// Data types/BACnet Enumerations/E_BACNETUNIT
TYPE E_BACNETUNIT:
(
	BACnetUnit_Area_square_meters	:=	0	,
	BACnetUnit_Area_square_feet	:=	1	,
	BACnetUnit_Electrical_milliamperes	:=	2	,
	BACnetUnit_Electrical_amperes	:=	3	,
	BACnetUnit_Electrical_ohms	:=	4	,
	BACnetUnit_Electrical_volts	:=	5	,
	BACnetUnit_Electrical_kilovolts	:=	6	,
	BACnetUnit_Electrical_megavolts	:=	7	,
	BACnetUnit_Electrical_volt_amperes	:=	8	,
	BACnetUnit_Electrical_kilovolt_amperes	:=	9	,
	BACnetUnit_Electrical_megavolt_amperes	:=	10	,
	BACnetUnit_Electrical_volt_amperes_reactive	:=	11	,
	BACnetUnit_Electrical_kilovolt_amperes_reactive	:=	12	,
	BACnetUnit_Electrical_megavolt_amperes_reactive	:=	13	,
	BACnetUnit_Electrical_degrees_phase	:=	14	,
	BACnetUnit_Electrical_power_factor	:=	15	,
	BACnetUnit_Energy_joules	:=	16	,
	BACnetUnit_Energy_kilojoules	:=	17	,
	BACnetUnit_Energy_watt_hours	:=	18	,
	BACnetUnit_Energy_kilowatt_hours	:=	19	,
	BACnetUnit_Energy_btus	:=	20	,
	BACnetUnit_Energy_therms	:=	21	,
	BACnetUnit_Energy_ton_hours	:=	22	,
	BACnetUnit_Enthalpy_joules_per_kilogram_dry_air	:=	23	,
	BACnetUnit_Enthalpy_btus_per_pound_dry_air	:=	24	,
	BACnetUnit_Frequency_cycles_per_hour	:=	25	,
	BACnetUnit_Frequency_cycles_per_minute	:=	26	,
	BACnetUnit_Frequency_hertz	:=	27	,
	BACnetUnit_Humidity_grams_of_water_per_kilogram_dry_air	:=	28	,
	BACnetUnit_Humidity_percent_relative_humidity	:=	29	,
	BACnetUnit_Length_millimeters	:=	30	,
	BACnetUnit_Length_meters	:=	31	,
	BACnetUnit_Length_inches	:=	32	,
	BACnetUnit_Length_feet	:=	33	,
	BACnetUnit_Light_watts_per_square_foot	:=	34	,
	BACnetUnit_Light_watts_per_square_meter	:=	35	,
	BACnetUnit_Light_lumens	:=	36	,
	BACnetUnit_Light_luxes	:=	37	,
	BACnetUnit_Light_foot_candles	:=	38	,
	BACnetUnit_Mass_kilograms	:=	39	,
	BACnetUnit_Mass_pounds_mass	:=	40	,
	BACnetUnit_Mass_tons	:=	41	,
	BACnetUnit_MassFlow_kilograms_per_second	:=	42	,
	BACnetUnit_MassFlow_kilograms_per_minute	:=	43	,
	BACnetUnit_MassFlow_kilograms_per_hour	:=	44	,
	BACnetUnit_MassFlow_pounds_mass_per_minute	:=	45	,
	BACnetUnit_MassFlow_pounds_mass_per_hour	:=	46	,
	BACnetUnit_Power_watts	:=	47	,
	BACnetUnit_Power_kilowatts	:=	48	,
	BACnetUnit_Power_megawatts	:=	49	,
	BACnetUnit_Power_btus_per_hour	:=	50	,
	BACnetUnit_Power_horsepower	:=	51	,
	BACnetUnit_Power_tons_refrigeration	:=	52	,
	BACnetUnit_Pressure_pascals	:=	53	,
	BACnetUnit_Pressure_kilopascals	:=	54	,
	BACnetUnit_Pressure_bars	:=	55	,
	BACnetUnit_Pressure_pounds_force_per_square_inch	:=	56	,
	BACnetUnit_Pressure_centimeters_of_water	:=	57	,
	BACnetUnit_Pressure_inches_of_water	:=	58	,
	BACnetUnit_Pressure_millimeters_of_mercury	:=	59	,
	BACnetUnit_Pressure_centimeters_of_mercury	:=	60	,
	BACnetUnit_Pressure_inches_of_mercury	:=	61	,
	BACnetUnit_Temperature_degrees_Celsius	:=	62	,
	BACnetUnit_Temperature_degrees_Kelvin	:=	63	,
	BACnetUnit_Temperature_degrees_Fahrenheit	:=	64	,
	BACnetUnit_Temperature_degree_days_Celsius	:=	65	,
	BACnetUnit_Temperature_degree_days_Fahrenheit	:=	66	,
	BACnetUnit_Time_years	:=	67	,
	BACnetUnit_Time_months	:=	68	,
	BACnetUnit_Time_weeks	:=	69	,
	BACnetUnit_Time_days	:=	70	,
	BACnetUnit_Time_hours	:=	71	,
	BACnetUnit_Time_minutes	:=	72	,
	BACnetUnit_Time_seconds	:=	73	,
	BACnetUnit_Velocity_meters_per_second	:=	74	,
	BACnetUnit_Velocity_kilometers_per_hour	:=	75	,
	BACnetUnit_Velocity_feet_per_second	:=	76	,
	BACnetUnit_Velocity_feet_per_minute	:=	77	,
	BACnetUnit_Velocity_miles_per_hour	:=	78	,
	BACnetUnit_Volume_cubic_feet	:=	79	,
	BACnetUnit_Volume_cubic_meters	:=	80	,
	BACnetUnit_Volume_imperial_gallons	:=	81	,
	BACnetUnit_Volume_liters	:=	82	,
	BACnetUnit_Volume_us_gallons	:=	83	,
	BACnetUnit_VolumetricFlow_cubic_feet_per_minute	:=	84	,
	BACnetUnit_VolumetricFlow_cubic_meters_per_second	:=	85	,
	BACnetUnit_VolumetricFlow_imperial_gallons_per_minute	:=	86	,
	BACnetUnit_VolumetricFlow_liters_per_second	:=	87	,
	BACnetUnit_VolumetricFlow_liters_per_minute	:=	88	,
	BACnetUnit_VolumetricFlow_us_gallons_per_minute	:=	89	,
	BACnetUnit_Other_degrees_angular	:=	90	,
	BACnetUnit_Other_degrees_Celsius_per_hour	:=	91	,
	BACnetUnit_Other_degrees_Celsius_per_minute	:=	92	,
	BACnetUnit_Other_degrees_Fahrenheit_per_hour	:=	93	,
	BACnetUnit_Other_degrees_Fahrenheit_per_minute	:=	94	,
	BACnetUnit_Other_no_units	:=	95	,
	BACnetUnit_Other_parts_per_million	:=	96	,
	BACnetUnit_Other_parts_per_billion	:=	97	,
	BACnetUnit_Other_percent	:=	98	,
	BACnetUnit_Other_percent_per_second	:=	99	,
	BACnetUnit_Other_per_minute	:=	100	,
	BACnetUnit_Other_per_second	:=	101	,
	BACnetUnit_Other_psi_per_degree_Fahrenheit	:=	102	,
	BACnetUnit_Other_radians	:=	103	,
	BACnetUnit_Other_revolutions_per_minute	:=	104	,
	BACnetUnit_Currency_currency1	:=	105	,
	BACnetUnit_Currency_currency2	:=	106	,
	BACnetUnit_Currency_currency3	:=	107	,
	BACnetUnit_Currency_currency4	:=	108	,
	BACnetUnit_Currency_currency5	:=	109	,
	BACnetUnit_Currency_currency6	:=	110	,
	BACnetUnit_Currency_currency7	:=	111	,
	BACnetUnit_Currency_currency8	:=	112	,
	BACnetUnit_Currency_currency9	:=	113	,
	BACnetUnit_Currency_currency10	:=	114	,
	BACnetUnit_Area_square_inches	:=	115	,
	BACnetUnit_Area_square_centimeters	:=	116	,
	BACnetUnit_Enthalpy_btus_per_pound	:=	117	,
	BACnetUnit_Length_centimeters	:=	118	,
	BACnetUnit_MassFlow_pounds_mass_per_second	:=	119	,
	BACnetUnit_Temperature_delta_degrees_Fahrenheit	:=	120	,
	BACnetUnit_Temperature_delta_degrees_Kelvin	:=	121	,
	BACnetUnit_Electrical_kilohms	:=	122	,
	BACnetUnit_Electrical_megohms	:=	123	,
	BACnetUnit_Electrical_millivolts	:=	124	,
	BACnetUnit_Energy_kilojoules_per_kilogram	:=	125	,
	BACnetUnit_Energy_megajoules	:=	126	,
	BACnetUnit_Entropy_joules_per_degree_Kelvin	:=	127	,
	BACnetUnit_Entropy_joules_per_kilogram_degree_Kelvin	:=	128	,
	BACnetUnit_Frequency_kilohertz	:=	129	,
	BACnetUnit_Frequency_megahertz	:=	130	,
	BACnetUnit_Frequency_per_hour	:=	131	,
	BACnetUnit_Power_milliwatts	:=	132	,
	BACnetUnit_Pressure_hectopascals	:=	133	,
	BACnetUnit_Pressure_millibars	:=	134	,
	BACnetUnit_VolumetricFlow_cubic_meters_per_hour	:=	135	,
	BACnetUnit_VolumetricFlow_liters_per_hour	:=	136	,
	BACnetUnit_Other_kilowatt_hours_per_square_meter	:=	137	,
	BACnetUnit_Other_kilowatt_hours_per_square_foot	:=	138	,
	BACnetUnit_Other_megajoules_per_square_meter	:=	139	,
	BACnetUnit_Other_megajoules_per_square_foot	:=	140	,
	BACnetUnit_Other_watts_per_square_meter_degree_kelvin	:=	141	,
	BACnetUnit_VolumetricFlow_cubic_feet_per_second	:=	142	,
	BACnetUnit_Other_percent_obscuration_per_foot	:=	143	,
	BACnetUnit_Other_percent_obscuration_per_meter	:=	144	,
	BACnetUnit_Electrical_milliohms	:=	145	,
	BACnetUnit_Energy_megawatt_hours	:=	146	,
	BACnetUnit_Energy_kilo_btus	:=	147	,
	BACnetUnit_Energy_mega_btus	:=	148	,
	BACnetUnit_Enthalpy_kilojoules_per_kilogram_dry_air	:=	149	,
	BACnetUnit_Enthalpy_megajoules_per_kilogram_dry_air	:=	150	,
	BACnetUnit_Entropy_kilojoules_per_degree_Kelvin	:=	151	,
	BACnetUnit_Entropy_megajoules_per_degree_Kelvin	:=	152	,
	BACnetUnit_Force_newton	:=	153	,
	BACnetUnit_MassFlow_grams_per_second	:=	154	,
	BACnetUnit_MassFlow_grams_per_minute	:=	155	,
	BACnetUnit_MassFlow_tons_per_hour	:=	156	,
	BACnetUnit_Power_kilo_btus_per_hour	:=	157	,
	BACnetUnit_Time_hundredths_seconds	:=	158	,
	BACnetUnit_Time_milliseconds	:=	159	,
	BACnetUnit_Torque_newton_meters	:=	160	,
	BACnetUnit_Velocity_millimeters_per_second	:=	161	,
	BACnetUnit_Velocity_millimeters_per_minute	:=	162	,
	BACnetUnit_Velocity_meters_per_minute	:=	163	,
	BACnetUnit_Velocity_meters_per_hour	:=	164	,
	BACnetUnit_VolumetricFlow_cubic_meters_per_minute	:=	165	,
	BACnetUnit_Acceleration_meters_per_second_per_second	:=	166	,
	BACnetUnit_Electrical_amperes_per_meter	:=	167	,
	BACnetUnit_Electrical_amperes_per_square_meter	:=	168	,
	BACnetUnit_Electrical_ampere_square_meters	:=	169	,
	BACnetUnit_Electrical_farads	:=	170	,
	BACnetUnit_Electrical_henrys	:=	171	,
	BACnetUnit_Electrical_ohm_meters	:=	172	,
	BACnetUnit_Electrical_siemens	:=	173	,
	BACnetUnit_Electrical_siemens_per_meter	:=	174	,
	BACnetUnit_Electrical_teslas	:=	175	,
	BACnetUnit_Electrical_volts_per_degree_Kelvin	:=	176	,
	BACnetUnit_Electrical_volts_per_meter	:=	177	,
	BACnetUnit_Electrical_webers	:=	178	,
	BACnetUnit_Light_candelas	:=	179	,
	BACnetUnit_Light_candelas_per_square_meter	:=	180	,
	BACnetUnit_Temperature_degrees_Kelvin_per_hour	:=	181	,
	BACnetUnit_Temperature_degrees_Kelvin_per_minute	:=	182	,
	BACnetUnit_Other_joule_seconds	:=	183	,
	BACnetUnit_Other_radians_per_second	:=	184	,
	BACnetUnit_Other_square_meters_per_Newton	:=	185	,
	BACnetUnit_Other_kilograms_per_cubic_meter	:=	186	,
	BACnetUnit_Other_newton_seconds	:=	187	,
	BACnetUnit_Other_newtons_per_meter	:=	188	,
	BACnetUnit_Other_watts_per_meter_per_degree_Kelvin	:=	189	,
	BACnetUnit_micro_siemens	:=	190	,
	BACnetUnit_cubic_feet_per_hour	:=	191	,
	BACnetUnit_us_gallons_per_hour	:=	192	,
	BACnetUnit_kilometers	:=	193	,
	BACnetUnit_micrometers	:=	194	,
	BACnetUnit_grams	:=	195	,
	BACnetUnit_milligrams	:=	196	,
	BACnetUnit_milliliters	:=	197	,
	BACnetUnit_milliliters_per_second	:=	198	,
	BACnetUnit_decibels	:=	199	,
	BACnetUnit_decibels_millivolt	:=	200	,
	BACnetUnit_decibels_volt	:=	201	,
	BACnetUnit_millisiemens	:=	202	,
	BACnetUnit_watt_hours_reactive	:=	203	,
	BACnetUnit_kilowatt_hours_reactive	:=	204	,
	BACnetUnit_megawatt_hours_reactive	:=	205	,
	BACnetUnit_millimeters_of_water	:=	206	,
	BACnetUnit_per_mille	:=	207	,
	BACnetUnit_grams_per_gram	:=	208	,
	BACnetUnit_kilograms_per_kilogram	:=	209	,
	BACnetUnit_grams_per_kilogram	:=	210	,
	BACnetUnit_milligrams_per_gram	:=	211	,
	BACnetUnit_milligrams_per_kilogram	:=	212	,
	BACnetUnit_grams_per_milliliter	:=	213	,
	BACnetUnit_grams_per_liter	:=	214	,
	BACnetUnit_milligrams_per_liter	:=	215	,
	BACnetUnit_micrograms_per_liter	:=	216	,
	BACnetUnit_grams_per_cubic_meter	:=	217	,
	BACnetUnit_milligrams_per_cubic_meter	:=	218	,
	BACnetUnit_micrograms_per_cubic_meter	:=	219	,
	BACnetUnit_nanograms_per_cubic_meter	:=	220	,
	BACnetUnit_grams_per_cubic_centimeter	:=	221	,
	BACnetUnit_becquerels	:=	222	,
	BACnetUnit_kilobecquerels	:=	223	,
	BACnetUnit_megabecquerels	:=	224	,
	BACnetUnit_gray	:=	225	,
	BACnetUnit_milligray	:=	226	,
	BACnetUnit_microgray	:=	227	,
	BACnetUnit_sieverts	:=	228	,
	BACnetUnit_millisieverts	:=	229	,
	BACnetUnit_microsieverts	:=	230	,
	BACnetUnit_microsieverts_per_hour	:=	231	,
	BACnetUnit_decibels_a	:=	232	,
	BACnetUnit_nephelometric_turbidity_unit	:=	233	,
	BACnetUnit_pH	:=	234	,
	BACnetUnit_grams_per_square_meter	:=	235	,
	BACnetUnit_minutes_per_degree_kelvin	:=	236
);
END_TYPE

// Global Variables/BACnet_Globals
{attribute 'Tc2GvlVarNames'}
VAR_GLOBAL
(* ADS read/write buffer for dynamic sized properties *)
	stBACnet_AdsBuffer		: ST_BACnet_GlobalAdsBuffer; (* 8kByte common ADS buffer used by function blocks that access BACnet over ADS *)
(* global linkable BACnet adapter *)
	fbBACnet_Adapter		: FB_BACnet_Adapter;
(* global visible BACnet adapter reference *)
	pBACnet_Adapter			: POINTER TO FB_BACnet_Adapter;
END_VAR
VAR_GLOBAL CONSTANT
(*********************************************
	Data field maximum
**********************************************)
	BACnet_MaxDayEntry			: UINT := 19;
	BACnet_MaxExSchEntries		: UINT := 9;
	BACnet_MaxTimeValues		: UINT := 9;
	BACnet_MaxObjIdList			: UINT := 1999;
	BACnet_MaxLogBufferEntries	: UINT := 499;
	BACnet_MaxDestinationArray	: UINT := 19;

(*********************************************
	error codes
**********************************************)
	BACnet_ERR_NO_ERROR				: UINT := 0;
	BACnet_ERR_NO_VALID_NET_ID		: UINT := 1;
	BACnet_ERR_WRONG_MAPPING		: UINT := 2;
	BACnet_ERR_OPERATIONAL			: UINT := 3;
	BACnet_ERR_NO_ETH_LINK			: UINT := 4;
	BACnet_ERR_NO_GATEWAY			: UINT := 5;
	BACnet_ERR_WOC_TRIGGER_UNSUP	: UINT := 6;
	BACnet_ERR_WOC_DISABLED			: UINT := 7;
	BACnet_ERR_INVALID_OBJECTID		: UINT := 8;
	BACnet_ERR_INVALID_OBJECTTYPE	: UINT := 10;
	BACnet_ERR_INVALID_CYCLETIME	: UINT := 11;
	BACnet_ERR_INVALID_PARAMETER	: UINT := 12;

(* errors with reset 20.. *)
	BACnet_ERR_PERSISTENT_WRITE		: UINT := 20;
	BACnet_ERR_INVALID_ADS_CONN		: UINT := 21;
	BACnet_ERR_CLIENT_TIMEOUT		: UINT := 22;
	BACnet_ERR_CLIENT_SERVICE		: UINT := 23;
	BACnet_ERR_WOC_TRIGGER_ACTIVE	: UINT := 24;
	BACnet_ERR_REVISION_READ		: UINT := 25;
	BACnet_ERR_PERSISTENT_PLC_WRITE	: UINT := 26;

(* ADS connection errors 30.. *)
	BACnet_ERR_ADS_NO_VALID_NET_ID	: UINT := 30; (* missing a valid Net ID *)
	BACnet_ERR_ADS_Data				: UINT := 31; (* ADS data length is wrong *)
	BACnet_ERR_ADS_Read				: UINT := 32; (* ADS read function was aborted *)
	BACnet_ERR_ADS_Write			: UINT := 33; (* ADS write function was aborted *)
	BACnet_ERR_ADS_ObjType			: UINT := 34; (* object type is wrong *)
	BACnet_ERR_ADS_ObjListEmpty		: UINT := 35; (* object list is empty *)
	BACnet_ERR_ADS_DeviceOP			: UINT := 36; (* device is not operational *)
	BACnet_ERR_ADS_NoDevice			: UINT := 37; (* no device object in object info list *)
	BACnet_ERR_ADS_ObjInstance		: UINT := 38; (* object list info is wrong *)
	BACnet_ERR_ADS_AmsPort			: UINT := 39; (* read AMS port is invalid (<1000) *)
	BACnet_ERR_ADS_ObjectId			: UINT := 40; (* object list info is wrong *)
	BACnet_ERR_ADS_LegacyStack		: UINT := 41; (* revision 6 stack detected (service is available from/above revision 9) *)
	BACnet_ERR_ADS_ObjIdMissmatch	: UINT := 42; (* object ID mapped and object list info are different *)
	BACnet_ERR_ADS_BufferSize		: UINT := 43; (* Property data larger than ADS buffer *)
	BACnet_ERR_ADS_SchedData		: UINT := 44; (* Wrong schedule property data *)
	BACnet_ERR_UnknownEventChoice	: UINT := 45; (* Unknown event choice type *)
	BACnet_ERR_UnknownEntryChoice	: UINT := 46; (* Unknown entry choice type *)
	BACnet_ERR_ADS_TooManyObjects	: UINT := 47; (* List of objects are longer than output list size *)
	BACnet_ERR_ADS_WrongEntrySize	: UINT := 48; (* expected entry size dosn't match read size *)
	BACnet_ERR_ADS_RecipientData	: UINT := 49; (* Invalid recipient data, device type expected *)
	BACnet_ERR_ADS_TooManyEntries	: UINT := 50; (* More entries than expected *)
	BACnet_ERR_ADS_NotEnoughEntries	: UINT := 51; (* Property incomplete, missing entries *)
	BACnet_ERR_ADS_Encoding			: UINT := 52; (* String encoding not supported *)
	BACnet_ERR_ADS_NoServerClient	: UINT := 53; (* Given ADS connection is not an server or client connection (expected bClient or bServer) *)
	BACnet_ERR_ADS_NoNotificationSink: UINT := 54; (* Given ADS connection is not an notification sink connection (expected bNSink) *)

(*********************************************
	other definitions
**********************************************)
	BACnet_ADSTimeOut			: TIME := t#15s;
	BACnet_PlcPersisTimeOut		: TIME := t#2m;
	BACnet_STRING_MAXLENGTH     : INT := 256;
	BACnet_ADSBufferSize		: INT := 8191; (* default 8kByte buffer *)

(* ADS index and groups *)
	BACnet_ADSIGRP_GET_OBJECT_LIST						: UDINT := 16#82400000;
	BACnet_ADSIGRP_CLIENT_COM_PARAMETER					: UDINT := 16#84000000;
	BACnet_ADSIGRP_DEV_R_GETADSPORTBYDEVID				: UDINT := 16#80000047; (* Get AMS Port BY Device ID *)
	BACnet_ADSIGRP_NTFSINK_EVENTNTF_CNT					: UDINT := 16#00000001;
	BACnet_ADSIGRP_NTFSINK_COVNTF_CNT					: UDINT := 16#00000002;
	BACnet_ADSIGRP_NTFSINK_EVENTNTF_READ				: UDINT := 16#00000003;
	BACnet_ADSIGRP_NTFSINK_COVNTF_READ					: UDINT := 16#00000004;
	BACnet_ADSIGRP_NTFSINK_EVENTNTF_DELETE				: UDINT := 16#00000005;
	BACnet_ADSIGRP_NTFSINK_COVNTF_DELETE				: UDINT := 16#00000006;
	BACnet_ADSIGRP_NTFSINK_EVENTNTF_INFO				: UDINT := 16#00000007;
	BACnet_ADSIGRP_NTFSINK_COVNTF_INFO					: UDINT := 16#00000008;
	BACnet_ADSIGRP_WRITE_NTFSINK_EVENTNTF_ACK			: UDINT := 16#00000009;
	BACnet_ADSIGRP_NTFSINK_W_EVENTNTF_ACK_BY_SEQUENCE	: UDINT := 16#0000000A;
	BACnet_ADSIGRP_NTFSINK_W_EVENTNTF_ACK_BY_PARAMETER	: UDINT := 16#0000000B;
	BACnet_ADSIGRP_NTFSINK_R_EVENTNTF_READ_BY_SEQUENCE	: UDINT := 16#0000000C;
	BACnet_ADSIGRP_NTFSINK_R_COVNTF_READ_BY_SEQUENCE	: UDINT := 16#0000000D;
	BACnet_ADSIGRP_NTFSINK_R_EVENTNTF_DELETE_BY_SEQUENCE: UDINT := 16#0000000E;
	BACnet_ADSIGRP_NTFSINK_R_COVNTF_DELETE_BY_SEQUENCE	: UDINT := 16#0000000F;


(* Object specifications *)
	arrBACnet_ObjectTypeNameShort : ARRAY[0..BACnetObjectType_ZCount] OF STRING(5) := [
		'AI' (* BACnetObjectType_AnalogInput :=0 *),
		'AO' (* BACnetObjectType_AnalogOutput :=1 *),
		'AV' (* BACnetObjectType_AnalogValue :=2 *),
		'BI' (* BACnetObjectType_BinaryInput :=3 *),
		'BO' (* BACnetObjectType_BinaryOutput :=4 *),
		'BV' (* BACnetObjectType_BinaryValue :=5 *),
		'CAL' (* BACnetObjectType_Calendar :=6 *),
		'CMD' (* BACnetObjectType_Command :=7 *),
		'DEV' (* BACnetObjectType_Device :=8 *),
		'EE' (* BACnetObjectType_EventEnrollment :=9 *),
		'FILE' (* BACnetObjectType_File :=10 *),
		'GROUP' (* BACnetObjectType_Group :=11 *),
		'LOOP' (* BACnetObjectType_Loop :=12 *),
		'MI' (* BACnetObjectType_MultiStateInput :=13 *),
		'MO' (* BACnetObjectType_MultiStateOutput :=14 *),
		'NC' (* BACnetObjectType_NotificationClass :=15 *),
		'PROG' (* BACnetObjectType_Program :=16 *),
		'SCHED' (* BACnetObjectType_Schedule :=17 *),
		'AVG' (* BACnetObjectType_Averaging :=18 *),
		'MV' (* BACnetObjectType_MultiStateValue :=19 *),
		'TLOG' (* BACnetObjectType_TrendLog :=20 *),
		'LP' (* BACnetObjectType_LifeSafetyPoint :=21 *),
		'LZ' (* BACnetObjectType_LifeSafetyZone :=22 *),
		'ACC' (* BACnetObjectType_Accumulator :=23 *),
		'PC' (* BACnetObjectType_PulseConverter :=24 *),
		''] (* BACnetObjectType_ZCount :=25 *);



END_VAR

// Version/Global_Version
// This function has been automatically generated from the project information.
VAR_GLOBAL CONSTANT
	{attribute 'const_non_replaced'}
	{attribute 'linkalways'}
	stLibVersion_Tc2_BACnetRev12 : ST_LibVersion := (iMajor := 2, iMinor := 4, iBuild := 3, iRevision := 0, sVersion := '2.4.3.0');
END_VAR

// POUs/[obsolete]/F_GetVersionTcBACnet
{attribute 'obsolete' := 'F_GetVersionTcBACnet is obsolete, use stLibVersion_Tc2_BACnetRev12 instead!'}
FUNCTION F_GetVersionTcBACnet : UINT		(* Gets the library version info *)
VAR_INPUT
	nVersionElement		: INT;
END_VAR


(* Possible nVersionElement number:
	1	:	major number
	2	:	minor number
	3	: 	revision number
*)

(* Version history:
Date		|	Version/Author			|	Created with				|	Remark
-----------------------------------------------------------------------------------------------------------------------------------
13/03/12	|	1.0.0	/ MAr			|	V2.11.0 (Build 2218)		|	* Renamed BACnet-datatype ENUM entries
20/03/12	|	1.1.0	/ MAr			|	V2.11.0 (Build 2219)		|	* Added new function blocks with ADS property write support (for WOC on local objects present_value)
			|							|								|	* Added optional input to FB_BACnet_Device to setup the valid ADS port (default 1000)
20/03/12	|	1.1.1	/ MAr			|	V2.11.0 (Build 2219)		|	* Removed obsolete flags in FB_BACnet_Program function block
27/03/12	|	1.1.2	/ MAr			|	V2.11.0 (Build 2219)		|	* FB_BACnet_ReadProp returns real processed data len (nProcessedLen)
			|							|								|	* new helper function "F_BACnet_GetObjId" added
28/03/12	|	1.1.3	/ MAr			|	V2.11.0 (Build 2219)		|	* fixed error reset in "FB_BACnet_Device"
			|							|								|	* filter object instance number in "F_BACnet_GetObjId" to prevent overflow
			|							|								|	* added ending element of BACnetObjectType-Enumeration
			|							|								|	* renamed "bErrorId" to "nErrorId" in "FB_BACnet_NotificationSinkDelEntry"
10/04/12	|	1.1.4	/ MAr			|	V2.11.0 (Build 2220)		|	* FB_BACnet_ReadProp extended with automatic handling for range properties (READ_RANGE)
21/05/12	|	1.2.0	/ MAr			|	V2.11.0 (Build 2222)		|	* Changed ENUM names to capital letter (upper case)
			|							|								|	* Renamed LOOP object process data "_SystemStatus" to "_PresentValueI"
			|							|								|	* Append update logic for remote device into remote object FBs (no need to call remote device FB explicit)
29/05/12	|	1.2.1	/ MAr			|	V2.11.0 (Build 2223)		|	* Append local object for Accumulator access (and also _EX version)
20/07/12	|	1.2.2	/ MAr			|	V2.11.0 (Build 2224)		|	* New kind of BACnet FBs "_RAW" for read/write raw values in PLC program instead of direct hardware link
			|							|								|	* Added "AckedTransitions" flags to "_EX" function blocks
			|							|								|	* Added automatic client reset to FB_BACnet_RemoteDevice (timeouts will counted, but didn't interrupt client functionality if auto-reset is active)
			|							|								|	* New time out counter as output status to FB_BACnet_RemoteDevice added
23/07/12	|	1.2.3	/ MAr			|	V2.11.0 (Build 2226)		|	* Added service fail counter to FB_BACnet_RemoteDevice
20/12/12	|	1.3.0	/ MAr	(Beta)	|	V2.11.0 (Build 2232)		|	* Added ADS-Connection blocks (easy to connect objects over ADS)
			|							|								|	* Added local object function blocks with revision 9 features (BETA versions!)
			|							|								|	* Major-change in exisiting object: FB_BACnet_Loop object dosn't write "OutOfService" anymore
			|							|								|	* New raw version of the ACC object type
			|							|								|	* Added flag helper functions
20/12/12	|	1.3.1	/ MAr	(Beta)	|	V2.11.0 (Build 2232)		|	* Optimized error handling for remote device
			|							|								|	* auto detect legacy mode in remote device and fill AdsConn infos from remote device inputs
08/07/13	|	1.3.2	/ MAr	(Beta)	|	V2.11.0 (Build 2234)		|	* added missing _RAW types to R9
21/08/13	|	1.3.3	/ MAr			|	V2.11.0 (Build 2234)		|	* added new function block for time synchronization over BACnet (local time --> BACnet server --> BACnet broadcast)
06/09/13	|	2.0.0	/ MAr			|	V2.11.0 (Build 2234)		|	* removed legacy function blocks and replaced with R9 versions
			|							|								|	* added function blocks for property access
			|							|								|	* error codes are complete global now
			|							|								|	* optimized process data (removed object ID for basic FBs, sorted process data with focus on alignment)
10/09/13	|	2.0.1	/ MAr			|	V2.11.0 (Build 2237)		|	* new function block for EE object add
02/10/13	|	2.0.2	/ MAr			|	V2.11.0 (Build 2237)		|	* Mapped LocalTime and -Date into Device object
			|							|								|	* Added some helper and signal functions
			|							|								|	* PID auto tuning added into LOOP_EX version
			|							|								|	* Added LOOP objects using internal stack LOOP controller (performance optimized)
			|							|								|	* Removed obsolete function blocks
05/11/13	|	2.0.3	/ MAr			|	V2.11.0 (Build 2237)		|	* Added Multi-State objects as RAW-type
			|							|								|	* Renamed BACnetInfo structure member
			|							|								|	* Added feedback and error flag to RAW function blocks
			|							|								|	* First cycle flag moved on first position in function block logic
			|							|								|	* added WOC-disable service and PLC-startup flag into device object
			|							|								|	* clear data buffer in ReadProp function block (because client data optimized and size of read data maybe lower than buffer size)
19/03/14	|	2.0.4	/ MAr			|	V2.11.0 (Build 2240)		|	* removed obsolete check
10/04/14	|	2.1.0	/ MAr			|	V2.11.0 (Build 2241)		|	* PLC ready flag delayed by device status
23/04/14	|	2.2.0	/ MAr			|	V2.11.0 (Build 2241)		|	* Removed "POLL" version of remote FBs (poll mode can be configured by function block comments)
			|							|								|	* Changed default present_value of object function blocks to "do-nothing"
			|							|								|	  (NULL is furthermore writeable by F_BACnet_RealNull or special Binary-PV [2] or multi-state [0] values)
			|							|								|	* Added new function blocks for PV values (F_BACnet_AnalogPV and F_BACnet_MultiStatePV)
			|							|								|	* Added "a-life" bit to remote device function block
20/05/14	|	2.2.1	/ MAr			|	V2.11.0 (Build 2241)		|	* Fixed "ReadMessageTexts"
			|							|								|	* Default value for command object changed to 0x0 instead 0xffffffff
02/06/14	|	2.2.2	/ MAr			|	V2.11.0 (Build 2241)		|	* Added Notification-Sink read and remove functions (Rev. 12 and above only)
			|							|								|	* Added Notification-Sink function block
			|							|								|	* optimized encoding function (when source and target are diffent memory areas with same byte size)
11/06/14	|	2.2.3	/ MAr			|	V2.11.0 (Build 2241)		|	* Added "bReload" input into local and remote device object
			|							|								|	* automatic LOOP mode detection (ideal mode vs. standard mode) according to the property unit of integral_ and derivative_constant
			|							|								|		- ideal mode means: clear parallel junktion of P, I and D (parameter Kp, Ki and Kd are gain [1] constants for each element)
			|							|								|		- standard mode means: serial junktion of P and I parallel to P and D (parameter Kp is the gain constant [1], Ti and Td are time based [s])
14/11/14	|	2.2.4	/ MAr			|	V2.11.0 (Build 2245)		|	* Added stValidFields into Notification-Event structure
			|							|								|	* Optimized STRING conversion for Object-ID and Date/Time
			|							|								|	* Optimized result type for F_BACnet_GetObjId
20/11/14	|	2.2.5	/ MAr			|	V2.11.0 (Build 2245)		|	* Optimized data handling for Log_Buffer property function block
05/12/14	|	2.2.6	/ MAr			|	V2.11.0 (Build 2245)		|	* Optimized process data default value for remote program object
16/01/15	|	2.2.7	/ MAr			|	V2.11.0 (Build 2245)		|	* New function for "Nothing" process data coding for analog* objects
19/01/15	|	2.3.0	/ MAr			|	V2.11.0	(Build 2245)		|	* Changed default FB to read-only (except local LOOP and PROG)
			|							|								|	* Append new "_WR" function block types to enable write access for commandable basic function blocks (remote and local)
23/01/15	|	2.3.1	/ MAr			|	V2.11.0	(Build 2245)		|	* Optimize value compare in ADS-type of analog* objects
10/02/15	|	2.4.0	/ MAr			|	V2.11.0	(Build 2245)		|	* Remove local _WR-Object types
23/10/15	|	2.4.1	/ MAr			|	V2.11.0 (Build 2248)		|	* Added exception- and weekly-schedule property with REAL value capability
04/11/15	|	2.4.2	/ MAr			|	V2.11.0 (Build 2248)		|	* Fixed data type handling in new REAL type properties
06/11/15	|	2.4.3	/ MAr			|	V2.11.0 (Build 2248)		|	* Fallback for PID mode, if property I or D is deactivated
*)

CASE nVersionElement OF
	1:	F_GetVersionTcBACnet := stLibVersion_Tc2_BACnetRev12.iMajor;
	2:	F_GetVersionTcBACnet := stLibVersion_Tc2_BACnetRev12.iMinor;
	3:	F_GetVersionTcBACnet := stLibVersion_Tc2_BACnetRev12.iBuild;
	4:	F_GetVersionTcBACnet := stLibVersion_Tc2_BACnetRev12.iRevision;
	ELSE
		F_GetVersionTcBACnet := 16#FFFF;
END_CASE

END_FUNCTION

// POUs/BACnet Objects/Local (Server)/FB_BACnet_Device
FUNCTION_BLOCK FB_BACnet_Device
VAR_INPUT
	bReset				: BOOL; (* reset errors *)
	bSupportBackup		: BOOL; (* support backup of PLC persistent data when BACnet backup service is used *)
	bWritePersis		: BOOL; (* Manual trigger for PLC and BACnet persistent data storage *)
	bDisableWOC			: BOOL; (* Deactivate write-on-change mechanism *)
	bReload				: BOOL; (* Reload ADS connection and increase reload counter (trigger autoget) *)
	nAmsPort			: T_AmsPort := 1000; (* default port when port can not be determined automatically *)
END_VAR
VAR_OUTPUT
	nRevision			: DINT := -1; (* protocol revision no. *)
	stAdsConn			: ST_BACnet_AdsConnection;
	eSystemStatus		: E_BACNETDEVICESTATUS;
	bBackupActive		: BOOL;
	bWritePersisActive	: BOOL;
	bOperational		: BOOL;
	bWOCDisabled		: BOOL;
	bFirstCycle			: BOOL;
	dtLocalTime			: ST_BACnet_DateTime;
	bError				: BOOL;
	nErrorId			: UINT;
END_VAR
VAR
	_ObjectId			AT%I*: DWORD;	(* ~(BACnet_ObjectIdentifier:		: LINK) *)
	_LocalDate			AT%I*: DWORD;	(* ~(BACnet_LocalDate		:		: LINK) *)
	_LocalTime			AT%I*: DWORD;	(* ~(BACnet_LocalTime		:		: LINK) *)
	_SystemStatus		AT%I*: WORD;	(* ~(BACnet_SystemStatus	:		: )
								   			(BACnet_ObjectType		: DEV	: )	*)
	_ServerStatus		AT%I*: WORD;	(* ~(BACnet_ServerStatus	:		: )	*)
	_ServerControl		AT%Q*: WORD;	(* ~(BACnet_ServerControl	:		: )	*)
	_fbWritePersistent	: FB_WritePersistentData;
	_rtrigBackup		: R_TRIG;
	_rtrigReset			: R_TRIG;

	_bHasStarted		: BOOL := TRUE;
	_nPlcPort			: T_AmsPort;

	_nUpdateCount	 	: UDINT := 0;
	_nUpdateCountAdp 	: UDINT := 0;
	_BACnetAdapter		: POINTER TO FB_BACnet_Adapter;
	_AdsConn			: _FB_BACnet_AdsConn;
	_WritePersistentProp: FB_BACnet_WriteProp;
	_ReadPersistentProp	: FB_BACnet_ReadProp;
	_iPersis			: INT;
	_nPersistentState	: DWORD;
	_ePersistentState	: E_BACNETPERSISTENTDATASTATE;
	_tonPersisTimeout	: TON;
	_tonPersisPoll		: TON;
	_bPersisWritten		: BOOL;
	_ReadRevisionProp	: FB_BACnet_ReadProp;
	_iRevision			: INT;
	_pLocalDate			: POINTER TO ST_BACnet_Date;
	_pLocalTime			: POINTER TO ST_BACnet_Time;
END_VAR

(* check pointer to bacnet adapter instance *)
IF pBACnet_Adapter > 0 THEN
	_BACnetAdapter := pBACnet_Adapter;
ELSE
	_BACnetAdapter := ADR(fbBACnet_Adapter);
END_IF

(* update adapter *)
IF _BACnetAdapter^._nUpdateCount = _nUpdateCountAdp THEN
	_BACnetAdapter^();
END_IF
(* remind current number of update counter *)
_nUpdateCountAdp := _BACnetAdapter^._nUpdateCount;

(* convert SystemStatus to enumeration *)
eSystemStatus := TO_INT(_SystemStatus);

(* reset trigger *)
_rtrigReset(CLK:= bReset, Q=> );
(* reset error ID and flag *)
IF (nErrorId < 20) OR (nErrorId >= 30) OR _rtrigReset.Q THEN
	nErrorId := BACnet_ERR_NO_ERROR;
END_IF

(* check if NetID is plausible *)
IF _BACnetAdapter^.sAmsNetId = '' THEN
	(* NetId not OK, return with error *)
	nErrorId := BACnet_ERR_NO_VALID_NET_ID;
END_IF

IF ((bSupportBackup) OR (_fbWritePersistent.START AND (_iPersis = 0))) THEN
	(* PLC can be backup't *)
	_ServerControl.0 := TRUE;
ELSE
	(* don't support PLC backup *)
	_ServerControl.0 := FALSE;
	_ServerControl.1 := FALSE;
END_IF

(* trigger backup flag *)
_rtrigBackup(CLK:= (eSystemStatus = BACnetDeviceStatus_BackupInProgress) AND (_iPersis = 0), Q=> );
IF (_iPersis = 0) THEN
	(* only backup if persistent state machine is idle *)
	IF _rtrigBackup.Q AND _ServerControl.0 THEN
		(* trigger backup function *)
		_fbWritePersistent.START := TRUE;
	ELSIF _fbWritePersistent.START AND (NOT _fbWritePersistent.BUSY) THEN
		IF _fbWritePersistent.ERR THEN
			(* backup aborted *)
			nErrorId := BACnet_ERR_PERSISTENT_PLC_WRITE;
		ELSE
			(* backup was successful *)
			_ServerControl.1 := TRUE;
		END_IF
	ELSIF (eSystemStatus <> BACnetDeviceStatus_BackupInProgress) THEN
		(* backup process finished *)
		_ServerControl.1 := FALSE;
	END_IF
END_IF

(* calculate PLC runtime port *)
_nPlcPort := TwinCAT_SystemInfoVarList._AppInfo.AdsPort;

(* call persistent backup *)
_fbWritePersistent(
	NETID	:= '',
	PORT	:= _nPlcPort,
	START	:= ,
	TMOUT	:= BACnet_PlcPersisTimeOut,
	MODE	:= SPDM_VAR_BOOST,
	BUSY	=> ,
	ERR		=> ,
	ERRID	=>
);

(* call ADS connection *)
IF (_ObjectId <> 16#00000000) THEN
	_AdsConn(
		bAutoReload		:= bOperational,
		bReload			:= 	(bReset AND (NOT _AdsConn.bReady))
						OR	bReload,
		bDevOperational	:= bOperational,
		sAmsNetId		:= _BACnetAdapter^.sAmsNetId,
		tDevObjId		:= _ObjectId,
		bIsClient		:= FALSE,
		bReady			=> ,
		bBusy			=> ,
		bDone			=> ,
		bError			=> ,
		nErrorId		=> ,
		stBACnetAds		=> );
END_IF

(* error when ADS connection failed *)
IF _AdsConn.bError THEN
	IF (_AdsConn.nErrorId = BACnet_ERR_ADS_LegacyStack) THEN
		nRevision := 6;
		stAdsConn.bServer := TRUE;
		stAdsConn.bClient := FALSE;
		IF		(NOT stAdsConn.bValid)
			OR	(stAdsConn.nDeviceId <> F_BACnet_GetObjInstance(_ObjectId))
			OR	(stAdsConn.nAmsPort <> nAmsPort)
			OR	(stAdsConn.sAmsNetId <> _BACnetAdapter^.sAmsNetId)
		THEN
			stAdsConn.nReload := stAdsConn.nReload + 1;
		END_IF
		stAdsConn.nDeviceId	:= F_BACnet_GetObjInstance(_ObjectId);
		stAdsConn.sAmsNetId	:= _BACnetAdapter^.sAmsNetId;
		stAdsConn.nAmsPort	:= nAmsPort;
		stAdsConn.bValid	:= TRUE;
	ELSE
		IF (nErrorId = 0) THEN
			nErrorId	:= _AdsConn.nErrorId;
		END_IF
		nRevision := -1;
		stAdsConn	:= _AdsConn.stBACnetAds;
	END_IF
ELSIF _AdsConn.bDone THEN
	stAdsConn := _AdsConn.stBACnetAds;
ELSIF (NOT _AdsConn.bReady) THEN
	nRevision := -1;
END_IF

(* read revision no. *)
_ReadRevisionProp(
	BACnetDevicePort:= stAdsConn.nAmsPort,
	bExecute		:= ,
	sNetId			:= stAdsConn.sAmsNetId,
	ObjectType		:= BACnetObjectType_Device,
	PropertyID		:= BACnetPropertyIdentifier_ProtocolRevision,
	DataType		:= BACnetDataType_UnsignedInteger,
	ObjectInstance	:= stAdsConn.nDeviceId,
	ptrValue		:= ADR(nRevision),
	nLenValue		:= SIZEOF(nRevision),
	bDone			=> ,
	bBusy			=> ,
	bError			=> ,
	nErrID			=> ,
	nProcessedLen	=> );

CASE _iRevision OF

	0: (* idle *)
		IF _AdsConn.bDone THEN
			IF stAdsConn.bValid THEN
				_iRevision := 1;
			END_IF
		END_IF
		_ReadRevisionProp.bExecute := FALSE;

	1: (* read property *)
		IF		_ReadRevisionProp.bExecute
			AND	(NOT _ReadRevisionProp.bBusy)
		THEN
			IF _ReadRevisionProp.bError THEN
				nErrorId := BACnet_ERR_REVISION_READ;
			END_IF
			_ReadRevisionProp.bExecute := FALSE;
			_iRevision := 0;
		ELSE
			_ReadRevisionProp.bExecute := TRUE;
		END_IF

END_CASE


(* Handle persistent data backup *)
_nPersistentState := TO_WORD(_ePersistentState);
_ReadPersistentProp(
	BACnetDevicePort:= stAdsConn.nAmsPort,
	bExecute		:= ,
	sNetId			:= stAdsConn.sAmsNetId,
	ObjectType		:= BACnetObjectType_Device,
	PropertyID		:= 516,
	DataType		:= BACnetDataType_PersistentDataState,
	ObjectInstance	:= F_BACnet_GetObjInstance(_ObjectId),
	ptrValue		:= ADR(_nPersistentState),
	nLenValue		:= SIZEOF(_nPersistentState),
	bDone			=> ,
	bBusy			=> ,
	bError			=> ,
	nErrID			=> ,
	nProcessedLen	=> );

_WritePersistentProp(
	BACnetDevicePort:= stAdsConn.nAmsPort,
	bExecute		:= ,
	sNetId			:= stAdsConn.sAmsNetId,
	ObjectType		:= BACnetObjectType_Device,
	PropertyID		:= 516,
	Priority		:= ,
	DataType		:= BACnetDataType_PersistentDataState,
	ObjectInstance	:= F_BACnet_GetObjInstance(_ObjectId),
	ptrValue		:= ADR(_nPersistentState),
	nLenValue		:= SIZEOF(_nPersistentState),
	bDone			=> ,
	bBusy			=> ,
	bError			=> ,
	nErrID			=> );
_ePersistentState := UDINT_TO_INT(_nPersistentState AND 16#0000FFFF);

CASE _iPersis OF
	0: (* idle *)
		IF		bWritePersis
			AND	(NOT bBackupActive)
			AND	(eSystemStatus <> BACnetDeviceStatus_BackupInProgress)
			AND	(nErrorId = BACnet_ERR_NO_ERROR)
		THEN
			IF stAdsConn.bValid THEN
				_iPersis := 1;
			ELSE
				nErrorId := BACnet_ERR_INVALID_ADS_CONN;
			END_IF
		END_IF
		_ReadPersistentProp.bExecute := FALSE;
		_WritePersistentProp.bExecute := FALSE;
		_bPersisWritten := FALSE;

	1: (* read persistent state machine *)
		IF _ReadPersistentProp.bExecute THEN
			IF _ReadPersistentProp.bError THEN
				_iPersis := 100;
				nErrorId := BACnet_ERR_PERSISTENT_WRITE;
				_ReadPersistentProp.bExecute := FALSE;
			ELSIF (NOT _ReadPersistentProp.bBusy) THEN
				_iPersis := 2;
				_ReadPersistentProp.bExecute := FALSE;
			END_IF
		ELSE
			_ReadPersistentProp.bExecute := TRUE;
		END_IF

	2: (* check state *)
		_tonPersisTimeout.IN := FALSE;
		_tonPersisPoll.IN := FALSE;

		IF _tonPersisPoll.Q THEN
			(* rescan state machine *)
			_iPersis := 1;

		ELSIF _tonPersisTimeout.Q THEN
			(* timeout *)
			_iPersis := 100;
			nErrorId := BACnet_ERR_PERSISTENT_WRITE;

		ELSIF (_ePersistentState = BACnetPersistentData_Disabled) THEN
			_iPersis := 10;

		ELSIF	(_ePersistentState = BACnetPersistentData_Initialize)
			OR	(_ePersistentState >= BACnetPersistentData_Write)
		THEN
			(* wait on idle state *)
			_tonPersisTimeout.IN := TRUE;
			_tonPersisPoll.IN := TRUE;

		ELSIF (_ePersistentState = BACnetPersistentData_NoChange) THEN
			(* start writing PLC *)
			_iPersis := 10;

		ELSIF (_ePersistentState = BACnetPersistentData_Ready) THEN
			IF _bPersisWritten THEN
				(* start writing PLC *)
				_iPersis := 10;
			ELSE
				(* start writing BACnet *)
				_iPersis := 3;
			END_IF

		ELSE
			(* wrong state *)
			_iPersis := 100;
			nErrorId := BACnet_ERR_PERSISTENT_WRITE;
		END_IF
		(* call timer *)
		_tonPersisTimeout(PT:= t#60s, Q=> , ET=> );
		_tonPersisPoll(PT:= t#2s, Q=> , ET=> );

	3: (* write BACnet persistent data *)
		IF _WritePersistentProp.bExecute THEN
			IF _WritePersistentProp.bError THEN
				nErrorId := BACnet_ERR_PERSISTENT_WRITE;
				_iPersis := 100;
				_WritePersistentProp.bExecute := FALSE;
			ELSIF (NOT _WritePersistentProp.bBusy) THEN
				_iPersis := 10; (* start writing PLC *)
				_WritePersistentProp.bExecute := FALSE;
				_bPersisWritten := TRUE;
			END_IF
		ELSE
			_WritePersistentProp.bExecute := TRUE;
			_ePersistentState := BACnetPersistentData_Write;
		END_IF

	10: (* write PLC persistent data *)
		IF _fbWritePersistent.START THEN
			IF _fbWritePersistent.ERR THEN
				(* Aborted *)
				nErrorId := BACnet_ERR_PERSISTENT_PLC_WRITE;
				_iPersis := 100;
				_fbWritePersistent.START := FALSE;
			ELSIF (NOT _fbWritePersistent.BUSY) THEN
				(* Finished *)
				_iPersis := 100;
				_fbWritePersistent.START := FALSE;
			END_IF
		ELSE
			_fbWritePersistent.START := TRUE;
		END_IF

	100:
		IF (NOT bWritePersis) THEN
			_iPersis := 0;
		END_IF

END_CASE

(* control *)
(* Disable write-on-change *)
_ServerControl.2	:= bDisableWOC;
(* PLC running - process data valid *)
_ServerControl.11	:=	(NOT _bHasStarted)
					AND	bOperational;

(* state *)
bWritePersisActive := (_iPersis > 0) AND (_iPersis < 100);
bBackupActive := (eSystemStatus = BACnetDeviceStatus_BackupInProgress);
bOperational :=	(_BACnetAdapter^.eAdapterStatus > BACnetAdapterStatus_Init);
bWOCDisabled := (_ServerStatus AND 16#0004) = 16#0004;
_pLocalDate := ADR(_LocalDate);
_pLocalTime := ADR(_LocalTime);
dtLocalTime.stDate := _pLocalDate^;
dtLocalTime.stTime := _pLocalTime^;

(* update counter *)
IF (_nUpdateCount = 0) AND _bHasStarted THEN
	bFirstCycle := TRUE;
ELSE
	bFirstCycle := FALSE;
END_IF
_bHasStarted := FALSE;
_nUpdateCount := _nUpdateCount + 1;
bError := (nErrorId <> BACnet_ERR_NO_ERROR);

END_FUNCTION_BLOCK

// POUs/BACnet Helper/F_BACnet_GetObjInstance
FUNCTION F_BACnet_GetObjInstance : UDINT
VAR_INPUT
	nObjectId : DWORD;
END_VAR
VAR
END_VAR

F_BACnet_GetObjInstance := nObjectId AND 16#003FFFFF;

END_FUNCTION

// POUs/FB_BACnet_Adapter
FUNCTION_BLOCK FB_BACnet_Adapter
VAR_INPUT
END_VAR
VAR_OUTPUT
	eAdapterStatus		: E_BACNETADAPTERSTATUS;
	bEthLinkOk			: BOOL;
	bGatewayOk			: BOOL;
	sAmsNetId			: T_AmsNetId;
	bFirstCycle			: BOOL;
	bError				: BOOL;
	nErrorId			: UINT;
END_VAR
VAR
	_DeviceStatus	AT%I*: WORD; (* ~(BACnet_DeviceStatus : : ) *)
	_AmsNetId		AT%I*: ARRAY[0..5] OF BYTE; (* ~(BACnet_AmsNetId : : ) *)
	_bHasStarted	: BOOL := TRUE;
	_nUpdateCount	: UDINT := 0;
END_VAR

(* reset error ID *)
nErrorId	:= BACnet_ERR_NO_ERROR;
bError		:= FALSE;

(* update bacnet adapter pointer *)
pBACnet_Adapter := THIS;

(* convert _DeviceStatus to enumeration *)
eAdapterStatus := UINT_TO_INT(SHR((_DeviceStatus AND 16#FF00), 8));

(* update netid *)
UpdateNetID();

(* states *)
bEthLinkOk := (NOT _DeviceStatus.0);
bGatewayOk := (eAdapterStatus = BACnetAdapterStatus_Complete) AND bEthLinkOk;

(* update counter *)
IF (_nUpdateCount = 0) AND _bHasStarted THEN
	bFirstCycle := TRUE;
	_bHasStarted := FALSE;
ELSE
	bFirstCycle := FALSE;
END_IF
_nUpdateCount := _nUpdateCount +1;

ACTION UpdateNetID:
(* read NetId and convert to string *)
sAmsNetId := F_CreateAmsNetId(_AmsNetId);
(* check if it plausible *)
IF sAmsNetId = '0.0.0.0.0.0' THEN
	(* NetId not OK, return with error *)
	bError := TRUE;
	nErrorId := BACnet_ERR_NO_VALID_NET_ID;
	sAmsNetId := '';
END_IF
END_ACTION

END_FUNCTION_BLOCK

// POUs/BACnet ADS/Connection/_FB_BACnet_AdsConn
FUNCTION_BLOCK _FB_BACnet_AdsConn
VAR_INPUT
	bAutoReload			: BOOL := TRUE; (* TRUE --> reload on device operational state and other changes *)
	bReload				: BOOL; (* FALSE --> TRUE refresh information *)
	bIsClient			: BOOL; (* TRUE --> Connection with client device (remote server) *)
END_VAR
VAR_IN_OUT
	bDevOperational		: BOOL;
	sAmsNetId			: T_AmsNetId;
	tDevObjId			: T_BACnet_ObjectIdentifier;
END_VAR
VAR_OUTPUT
	bReady				: BOOL;
	bBusy				: BOOL;
	bDone				: BOOL;
	bError				: BOOL;
	nErrorId			: UINT;
	stBACnetAds			: ST_BACnet_AdsConnection;
END_VAR
VAR
	_BACnetAmsNetID		: T_AmsNetId;
	_fbAdsRead			: FW_AdsRead;
	_arrAdsBuf			: ARRAY[0..13] OF DWORD;
	_rtrigReload		: R_TRIG;
	_rtrigOP			: R_TRIG;
	_i					: INT;
	_nDevObjects		: UDINT;
	_nObjIdx			: UDINT;
	_nAmsPort			: UINT;
	_tObjId				: T_BACnet_ObjectIdentifier := 16#FFFFFFFF;
END_VAR

(*
#define ADSIGRP_BACNET_CLIENT_COM_PARAMETER                      0x010

typedef struct _BACnetDevComData
{
      BACnetObjectIdentifier deviceObjIdentifier;
      BACnetAddress                  netAddress;                      // 10 Byte
      WORD                                 UdpPort;
      DWORD                                IPadress;       
      WORD                                 maxApdu;                         // wird im "Iam" Frame gesetzt
      WORD                                 vendorId;                        // wird im "Iam" Frame gesetzt
      DWORD                                maxSegments;                     // 0 == unspecified number of segments
      DWORD                                segmentTimeout;            // wenn 0 dann Defaultwerte des Devices nehmen 
      DWORD                                apduTimeout;                     // wenn 0 dann Defaultwerte des Devices nehmen
      DWORD                                nApduRetries;              // wenn 0 dann Defaultwerte des Devices nehmen
      BYTE                                 ethernetMacAddr[6];   // Ethernet MAC Address
      BYTE                                 segmentsSupported;         // segmentation both, transmit, receive, no (0 == segmentation both)
      BYTE                                 reserved;
} BACnetDevComData, *PBACnetDevComData;

-----------------------------------------------------
Server:

AdsReadInd, IndexGroup:
#define ADSIGRP_BACNET_GET_OBJECT_LIST                                 0x009

indexOffset == 0 -> Anzahl der Objekte

gerader Index -> Objekttyp
ungerader Index -> ObjetInstanz

IndexOffset 2 sollte daher die DeviceID des Servers sein
*)

(* ads communication *)
_fbAdsRead(
	sNetId		:= _BACnetAmsNetID,
	nPort		:= ,
	nIdxGrp		:= ,
	nIdxOffs	:= ,
	cbReadLen	:= SIZEOF(_arrAdsBuf),
	pReadBuff	:= ADR(_arrAdsBuf),
	bExecute	:= ,
	tTimeout	:= BACnet_ADSTimeOut,
	bBusy		=> ,
	bError		=> ,
	nErrId		=> ,
	cbRead		=> );

(* catch reload event trigger *)
_rtrigReload(CLK:= bReload, Q=> );
_rtrigOP(CLK:= bDevOperational, Q=> );

(* state machine *)
CASE _i OF

	0: (* Idle *)
		IF sAmsNetId = '' THEN
			(* NetId not OK, return with error *)
			nErrorId := BACnet_ERR_ADS_NO_VALID_NET_ID;
			stBACnetAds.bValid := FALSE;
			_BACnetAmsNetID := '';
		ELSIF (F_BACnet_GetObjType(tDevObjId) <> BACnetObjectType_Device) THEN
			(* Object type is not device *)
			nErrorId := BACnet_ERR_ADS_ObjectId;
			stBACnetAds.bValid := FALSE;
			_tObjId := 0;
		ELSIF	_rtrigReload.Q
			OR	(		(		(sAmsNetId <> stBACnetAds.sAmsNetId)
							OR	(tDevObjId <> _tObjId)
							OR	(_BACnetAmsNetID <> sAmsNetId)
							OR	_rtrigOP.Q
						)
					AND	bAutoReload
				)
		THEN
			IF (NOT bDevOperational) THEN
				(* BACnet adapter error *)
				nErrorId := BACnet_ERR_ADS_DeviceOP;
				stBACnetAds.bValid := FALSE;
			ELSE
				nErrorId := BACnet_ERR_NO_ERROR;
				_i := 1;
				(* store connection info *)
				_BACnetAmsNetID	:= sAmsNetId;
				_tObjId := tDevObjId;
			END_IF
		END_IF
		bDone := FALSE;

	(* Determin the AMS port *)
	1:
		IF _fbAdsRead.bExecute THEN
			IF _fbAdsRead.bError THEN
				IF ((UDINT_TO_DWORD(_fbAdsRead.nErrId) AND 16#0000FFFF) = 16#0703) THEN
					(* couldn't read service for AMS port of the device - maybe R6 stack running *)
					nErrorId := BACnet_ERR_ADS_LegacyStack;
				ELSE
					nErrorId := BACnet_ERR_ADS_Read;
				END_IF
				_fbAdsRead.bExecute := FALSE;
				_i := 100;
				stBACnetAds.bValid := FALSE;
			ELSIF (NOT _fbAdsRead.bBusy) THEN
				_fbAdsRead.bExecute := FALSE;
				(* check if port info is valid *)
				IF (_fbAdsRead.cbRead = 2) THEN
					_nAmsPort := DWORD_TO_UINT(_arrAdsBuf[0] AND 16#0000FFFF);
					(* length ok? *)
					IF _nAmsPort >= 1000 THEN
						IF bIsClient THEN
							_i := 100;
							stBACnetAds.nDeviceId := F_BACnet_GetObjInstance(tDevObjId);
						ELSE
							_i := 11;
						END_IF
					ELSE
						(* wrong length, abort *)
						_i := 100;
						nErrorId := BACnet_ERR_ADS_AmsPort;
						stBACnetAds.bValid := FALSE;
					END_IF
				ELSE
					nErrorId := BACnet_ERR_ADS_Data;
					_i := 100;
					stBACnetAds.bValid := FALSE;
				END_IF
			END_IF
		ELSE
			(* start ADS reading *)
			_fbAdsRead.bExecute := TRUE;
			_fbAdsRead.nIdxGrp := BACnet_ADSIGRP_DEV_R_GETADSPORTBYDEVID;
			_fbAdsRead.nPort := 65535;
			_fbAdsRead.nIdxOffs := tDevObjId;
		END_IF

	(* try READ server info -object list length- *)
	11:
		IF _fbAdsRead.bExecute THEN
			IF _fbAdsRead.bError THEN
				_fbAdsRead.bExecute := FALSE;
				_i := 100;
				nErrorId := BACnet_ERR_ADS_Read;
				stBACnetAds.bValid := FALSE;
			ELSIF (NOT _fbAdsRead.bBusy) THEN
				_fbAdsRead.bExecute := FALSE;
				(* check if object list is valid *)
				IF (_fbAdsRead.cbRead = 4) THEN
					_nDevObjects := _arrAdsBuf[0];
					(* length ok? *)
					IF _nDevObjects >= 1 THEN
						_i := 12;
						_nObjIdx := 0;
					ELSE
						(* wrong length, abort *)
						_i := 100;
						nErrorId := BACnet_ERR_ADS_ObjListEmpty;
						stBACnetAds.bValid := FALSE;
					END_IF
				ELSE
					nErrorId := BACnet_ERR_ADS_Data;
					_i := 100;
					stBACnetAds.bValid := FALSE;
				END_IF
			END_IF
		ELSE
			(* start ADS reading *)
			_fbAdsRead.bExecute := TRUE;
			_fbAdsRead.nIdxGrp := BACnet_ADSIGRP_GET_OBJECT_LIST;
			_fbAdsRead.nPort := _nAmsPort;
			_fbAdsRead.nIdxOffs := 0;
		END_IF

	(* try READ server info -object type- *)
	12:
		IF _fbAdsRead.bExecute THEN
			IF _fbAdsRead.bError THEN
				_fbAdsRead.bExecute := FALSE;
				_i := 100;
				nErrorId := BACnet_ERR_ADS_Read;
				stBACnetAds.bValid := FALSE;
			ELSIF (NOT _fbAdsRead.bBusy) THEN
				_fbAdsRead.bExecute := FALSE;
				(* check if type is valid *)
				IF (_fbAdsRead.cbRead = 4) THEN
					IF (_arrAdsBuf[0] = INT_TO_DWORD(BACnetObjectType_Device)) THEN
						(* device object found, go on *)
						_i := 13;
					ELSE
						(* wrong object type, next list entry *)
						_i := 12; (* remain in current step *)
						_nObjIdx := _nObjIdx + 1;
					END_IF
				ELSE
					nErrorId := BACnet_ERR_ADS_Data;
					_i := 100;
					stBACnetAds.bValid := FALSE;
				END_IF
			END_IF
		ELSE
			(* start ADS reading *)
			IF _nObjIdx < _nDevObjects THEN
				_fbAdsRead.bExecute := TRUE;
				_fbAdsRead.nIdxGrp := BACnet_ADSIGRP_GET_OBJECT_LIST;
				_fbAdsRead.nIdxOffs := (_nObjIdx * 2) + 2;
				_fbAdsRead.nPort := _nAmsPort;
			ELSE
				(* no device found, abort *)
				nErrorId := BACnet_ERR_ADS_NoDevice;
				_i := 100;
				stBACnetAds.bValid := FALSE;
			END_IF
		END_IF

	(* try READ server info -object instance- *)
	13:
		IF _fbAdsRead.bExecute THEN
			IF _fbAdsRead.bError THEN
				_fbAdsRead.bExecute := FALSE;
				_i := 100;
				nErrorId := BACnet_ERR_ADS_Read;
				stBACnetAds.bValid := FALSE;
			ELSIF (NOT _fbAdsRead.bBusy) THEN
				_fbAdsRead.bExecute := FALSE;
				(* preset done *)
				_i := 100;
				(* check if ID is valid *)
				IF (_fbAdsRead.cbRead = 4) THEN
					IF (_arrAdsBuf[0] <= 16#3FFFFF) THEN
						IF (F_BACnet_GetObjInstance(tDevObjId) = _arrAdsBuf[0]) THEN
							stBACnetAds.nDeviceId := F_BACnet_GetObjInstance(tDevObjId);
						ELSE
							nErrorId := BACnet_ERR_ADS_ObjIdMissmatch;
							stBACnetAds.bValid := FALSE;
						END_IF
					ELSE
						nErrorId := BACnet_ERR_ADS_ObjInstance;
						stBACnetAds.bValid := FALSE;
					END_IF
				ELSE
					nErrorId := BACnet_ERR_ADS_Data;
					stBACnetAds.bValid := FALSE;
				END_IF
			END_IF
		ELSE
			(* start ADS reading *)
			_fbAdsRead.bExecute := TRUE;
			_fbAdsRead.nIdxGrp := BACnet_ADSIGRP_GET_OBJECT_LIST;
			_fbAdsRead.nIdxOffs := (_nObjIdx * 2) + 1;
			_fbAdsRead.nPort := _nAmsPort;
		END_IF

	100: (* Done *)
		bDone := (nErrorId = BACnet_ERR_NO_ERROR);
		IF (NOT bDone) THEN
			stBACnetAds.bValid := FALSE;
		ELSE
			(* set states *)
			stBACnetAds.bServer := (NOT bIsClient);
			stBACnetAds.bClient := bIsClient;
			stBACnetAds.bValid := TRUE;
			(* count update *)
			stBACnetAds.nReload := stBACnetAds.nReload + 1;
		END_IF
		(* remind device AmsNetID and port *)
		stBACnetAds.sAmsNetId	:= _BACnetAmsNetID;
		stBACnetAds.nAmsPort	:= _nAmsPort;
		(* go idle *)
		_i := 0;

END_CASE

(* set error flag *)
bError	:= (nErrorId <> BACnet_ERR_NO_ERROR);
bBusy	:= _i > 0;
bReady	:= (NOT bError) AND ((NOT bBusy) OR bReady);

END_FUNCTION_BLOCK

// POUs/BACnet Helper/F_BACnet_GetObjType
FUNCTION F_BACnet_GetObjType : E_BACNETOBJECTTYPE
VAR_INPUT
	nObjectId : DWORD;
END_VAR
VAR
END_VAR

F_BACnet_GetObjType := TO_INT(SHR((nObjectId AND 16#FFC00000), 22));

END_FUNCTION

// POUs/BACnet ADS/Properties/Common/FB_BACnet_WriteProp
FUNCTION_BLOCK FB_BACnet_WriteProp
VAR_INPUT
	BACnetDevicePort	: UINT := 16#FFFF;
	bExecute			: BOOL;
	sNetId				: T_AmsNetId;
	ObjectType			: E_BACNETOBJECTTYPE;
	PropertyID			: E_BACNETPROPERTYIDENTIFIER;
	Priority			: E_BACNETPRIORITY;
	DataType			: E_BACNETDATATYPES;
	ObjectInstance		: UDINT;
	ptrValue			: POINTER TO BYTE;
	nLenValue			: UDINT; (* byte size of value (SIZEOF) *)
END_VAR
VAR_OUTPUT
	bDone				: BOOL;
	bBusy				: BOOL;
	bError				: BOOL;
	nErrID				: UDINT;
END_VAR
VAR
	_Write				: ADSWRITE;
	_rtrigStart			: R_TRIG;
	_len_data			: UDINT;
	_nPrio 				: UDINT;
	_ptrDWORD			: POINTER TO DWORD;
	_ptrREAL			: POINTER TO REAL;
	_ptrBYTE			: POINTER TO BYTE;
	_dataPointer		: POINTER TO BYTE;
	_dwordVal			: DWORD;
END_VAR

(* catch the start flag *)
	_rtrigStart(Clk:=bExecute);

(* prepare *)
	IF _rtrigStart.Q AND (NOT bBusy) THEN
		_Write(WRITE := FALSE);
		bDone := FALSE;
		bBusy := TRUE;
		bError := FALSE;
		nErrId := 0;
		_nPrio := SHL(INT_TO_UDINT(Priority), 26);
		_len_data := nLenValue; (* in default, take the user given length *)
		_dataPointer := ptrValue;
		CASE DataType OF
			BACnetDataType_Null 				: _len_data := 0; (* set length to zero *)
			BACnetDataType_Bool 				: _len_data := _len_data; (* 1 *)
			BACnetDataType_CharacterStringExt	: _len_data := _len_data; (* 2 *)

			BACnetDataType_UnsignedInteger,
			BACnetDataType_SignedInteger 		: _len_data := MIN(_len_data, 4); (* 4 *)
				IF (_len_data >= 4) THEN
					(* source data type bigger/equal 4 byte --> OK, take first 4 byte *)
					_ptrDWORD := ptrValue;
				ELSE
					(* upgrade data type from less 4 byte to fully double word *)
					_dwordVal := 0;
					_ptrDWORD := ADR(_dwordVal);
					MEMCPY(destAddr:=_ptrDWORD, srcAddr:=ptrValue, n:=_len_data);
					_dataPointer := _ptrDWORD; (* from here on, point to the internal data source *)
					_len_data := SIZEOF(_dwordVal); (* increase size to internal data type length *)
				END_IF
				(* make some plausibility checks *)
				IF	(		ObjectType = BACnetObjectType_MultiStateInput
						OR	ObjectType = BACnetObjectType_MultiStateOutput
						OR	ObjectType = BACnetObjectType_MultiStateValue
					)
				THEN
					IF _ptrDWORD^ = 0 THEN
						(* set data type and data length to NULL operation *)
						_len_data := 0;
					END_IF
				END_IF

			BACnetDataType_Real 				: _len_data := _len_data; (* 4 *)
				_ptrREAL := ptrValue;
				IF (NOT F_BACnet_IsFinite(_ptrREAL^)) THEN
					(* set data type and data length to NULL operation *)
					_len_data := 0;
				END_IF

			BACnetDataType_Double 				: _len_data := _len_data; (* 8 *)
			BACnetDataType_OctetString 			: _len_data := _len_data; (* 8 *)
			BACnetDataType_Enumerated 			: _len_data := _len_data; (* 8 *)
			BACnetDataType_LimitEnable			: _len_data := _len_data; (* 4 *)
			BACnetDataType_BitString 			: _len_data := _len_data; (* 11 *)

			BACnetDataType_BinaryPV				: _len_data := MIN(_len_data, 1); (* 1 *)
				_ptrByte := ptrValue;
				IF		_len_data <= 0
					OR	_ptrByte^ >= 2
				THEN
					_len_data := 0;
				END_IF
		END_CASE
	ELSIF (NOT bExecute) THEN
		bDone := FALSE;
	END_IF

(* execute *)
	IF bBusy THEN
		_Write(	NETID:= sNetId,
				PORT:= BACnetDevicePort,
				IDXGRP:=16#80000000 + INT_TO_UDINT(PropertyID) + _nPrio,
				IDXOFFS:= F_BACnet_GetObjId(ObjectType, ObjectInstance),
				LEN:= _len_data,
				SRCADDR:= _dataPointer,
				WRITE:= TRUE,
				TMOUT:= BACnet_ADSTimeOut);
		IF NOT _Write.Busy THEN
			IF _Write.Err THEN
				nErrID := _Write.ErrId;
				bError := TRUE;
			END_IF
			_Write(WRITE := FALSE);
			bBusy := FALSE;
			bDone := NOT bError;
		END_IF
	END_IF

END_FUNCTION_BLOCK

// POUs/BACnet Helper/Real/F_BACnet_IsFinite
FUNCTION F_BACnet_IsFinite : BOOL
VAR_INPUT
	fValue		: REAL;
END_VAR
VAR
	fArg		: T_Arg;
END_VAR

fArg.cbLen := SIZEOF(fValue);
fArg.eType := ARGTYPE_REAL;
fArg.pData := ADR(fValue);
F_BACnet_IsFinite := IsFinite(fArg);

END_FUNCTION

// POUs/BACnet Helper/F_BACnet_GetObjId
FUNCTION F_BACnet_GetObjId : T_BACnet_ObjectIdentifier
VAR_INPUT
	ObjectType		: E_BACNETOBJECTTYPE;
	ObjectInstance	: UDINT;
END_VAR
VAR
END_VAR

F_BACnet_GetObjId := F_BACnet_GetObjInstance(ObjectInstance) + SHL(INT_TO_UDINT(ObjectType), 22);

END_FUNCTION

// POUs/BACnet ADS/Properties/Common/FB_BACnet_ReadProp
FUNCTION_BLOCK FB_BACnet_ReadProp
VAR_INPUT
	BACnetDevicePort	: UINT := 16#FFFF;
	bExecute			: BOOL;
	sNetId				: T_AmsNetId;
	ObjectType			: E_BACNETOBJECTTYPE;
	PropertyID			: E_BACNETPROPERTYIDENTIFIER;
	DataType			: E_BACNETDATATYPES;
	ObjectInstance		: UDINT;
	ptrValue			: POINTER TO BYTE;
	nLenValue			: UDINT; (* byte size of value (SIZEOF) *)
END_VAR
VAR_OUTPUT
	bDone				: BOOL;
	bBusy				: BOOL;
	bError				: BOOL;
	nErrID				: UDINT;
	nProcessedLen		: UDINT; (* the received data length (can be different to given length) *)
END_VAR
VAR
	_Read				: FW_AdsRead;
	_rtrigStart			: R_TRIG;
	_len_data			: UDINT;
END_VAR

(* catch the start flag *)
	_rtrigStart(Clk:=bExecute);

(* prepare *)
	IF _rtrigStart.Q AND (NOT bBusy) THEN
		_Read(bExecute := FALSE);
		bDone := FALSE;
		bBusy := TRUE;
		bError := FALSE;
		nErrId := 0;
		nProcessedLen := 0;
		(* in default, take the user given length *)
		_len_data := nLenValue;
		(* set index group for read property access *)
		_Read.nIdxGrp := 16#80000000 + INT_TO_UDINT(PropertyID);
		(* handle special data type things *)
		CASE DataType OF
			BACnetDataType_Null 				: _len_data := 0; (* set length to zero *)
			BACnetDataType_Bool 				: _len_data := _len_data; (* 1 *)
			BACnetDataType_CharacterStringExt	: _len_data := _len_data; (* 2 *)
			BACnetDataType_UnsignedInteger 		: _len_data := _len_data; (* 4 *)
			BACnetDataType_SignedInteger 		: _len_data := _len_data; (* 4 *)
			BACnetDataType_Real 				: _len_data := _len_data; (* 4 *)
			BACnetDataType_Double 				: _len_data := _len_data; (* 8 *)
			BACnetDataType_OctetString 			: _len_data := _len_data; (* 8 *)
			BACnetDataType_Enumerated 			: _len_data := _len_data; (* 8 *)
			BACnetDataType_LimitEnable			: _len_data := _len_data; (* 4 *)
			BACnetDataType_BitString 			: _len_data := _len_data; (* 11 *)
			BACnetDataType_LogRecordList:
				_len_data := _len_data; (* n *)
				_Read.nIdxGrp := _Read.nIdxGrp + 16#03800000; (* read range *)
		END_CASE;
	ELSIF (NOT bExecute) THEN
		bDone := FALSE;
	END_IF


(* execute *)
	IF bBusy THEN
		_Read(
			sNetId		:= sNetId,
			nPort		:= BACnetDevicePort,
			nIdxGrp		:= , (* see above *)
			nIdxOffs	:= F_BACnet_GetObjId(ObjectType, ObjectInstance),
			cbReadLen	:= _len_data,
			pReadBuff	:= ptrValue,
			bExecute	:= TRUE,
			tTimeout	:= BACnet_ADSTimeOut,
			bBusy		=> ,
			bError		=> ,
			nErrId		=> ,
			cbRead		=> );
		IF (NOT _Read.bBusy) THEN
			IF _Read.bError THEN
				nErrID := _Read.nErrId;
				bError := TRUE;
				nProcessedLen := 0;
			ELSE
				(* success *)
				nProcessedLen := _Read.cbRead;
				IF (_Read.cbRead < nLenValue) THEN
					(* fill unused part of buffer with zero *)
					MEMSET(destAddr:=(ptrValue+_Read.cbRead), fillByte:=0, n:=(nLenValue-_Read.cbRead));
				END_IF
			END_IF
			_Read(bExecute := FALSE);
			bBusy := FALSE;
			bDone := NOT bError;
		END_IF;
	END_IF

END_FUNCTION_BLOCK

// POUs/BACnet Objects/Local (Server)/FB_BACnet_Program
FUNCTION_BLOCK FB_BACnet_Program
VAR_INPUT
	bRelease			: BOOL;
	bCommonError		: BOOL;
	bWaitForSomething	: BOOL;
	stDoneFlags			: ST_BACnet_ProgramHandshakeRequests;
	stFailedFlags		: ST_BACnet_ProgramHandshakeRequests;
	bModeUnloadComplex	: BOOL := TRUE;
END_VAR
VAR_IN_OUT
	Device				: FB_BACnet_Device;
END_VAR
VAR_OUTPUT
	bReady				: BOOL;
	bOverridden			: BOOL;
	bOutOfService		: BOOL;
	bFault				: BOOL;
	bInAlarm			: BOOL;
	stRequestFlags		: ST_BACnet_ProgramHandshakeRequests;
	stActiveStateFlags	: ST_BACnet_ProgramHandshakeStates;
	bError				: BOOL;
	nErrorId			: UINT;
END_VAR
VAR
(* from BACnet to PLC *)
	_ProgramChange AT%I*: WORD;			(* ~(BACnet_ProgramChange 				:		: )
											(BACnet_ObjectType 					: PROG	: ) *)
	_StatusFlags AT%I*: WORD;			(* ~(BACnet_StatusFlags 				:		: )	*)

(* from PLC to BACnet *)
	_ProgramState AT%Q*: WORD;			(* ~(BACnet_ProgramState 				:		: ) *)
	_ReasonForHalt AT%Q*: WORD;			(* ~(BACnet_ReasonForHalt 				:		: )	*)
	_SetProgramReadyState AT%Q*: BOOL;	(* ~(BACnet_SetProgramReadyState 		:		: )	*)

(* internal signals *)
	_StatusFlagsBits 	: ST_BACnet_StatusFlags;
	_bTriggerSetup		: BOOL;
	_ActiveChange		: E_BACNETPROGRAMREQUEST; (* ACTIVE PROGRAM CHANGE *)
	_bLockedForChange	: BOOL;
	_nUpdateCount		: UDINT := 0;
END_VAR

(* update server device *)
IF (Device._nUpdateCount = _nUpdateCount) THEN
	Device();
END_IF
(* remind current number of update counter *)
_nUpdateCount := Device._nUpdateCount;

(* check BitString format of StatusFlags --> if StatusFlags are less than 4, object isn't linked correctly *)
IF (_StatusFlags < 4) THEN
	(* wrong mapping *)
	nErrorId := BACnet_ERR_WRONG_MAPPING;
	bReady := FALSE;

ELSIF Device.bOperational THEN
	(* ready state *)
	bReady := TRUE;
	nErrorId := BACnet_ERR_NO_ERROR;

	(* decode status flags *)
	_StatusFlagsBits := F_BACnet_StatusFlags(_StatusFlags);

	(* copy states to output *)
	bOverridden := _StatusFlagsBits.overridden;
	bOutOfService := _StatusFlagsBits.out_of_service;
	bFault := _StatusFlagsBits.fault;
	bInAlarm := _StatusFlagsBits.in_alarm;

	(* execute change *)
	CASE _ActiveChange OF
		BACnetProgramRequest_ready:
			(* idle *);

		BACnetProgramRequest_load:
			_ProgramState	 := TO_WORD(BACnetProgramState_loading);
			_ActiveChange	:= BACnetProgramRequest_ready;

		BACnetProgramRequest_restart,
		BACnetProgramRequest_run:
			IF _bTriggerSetup THEN
				(* wait on setup finish *)
				IF stFailedFlags.bSetup OR bCommonError OR (NOT bRelease) THEN
					(* abort *)
					_ProgramState := TO_WORD(BACnetProgramState_halted);
					_ActiveChange := BACnetProgramRequest_ready;
					_ReasonForHalt  := TO_WORD(BACnetProgramError_progerror_internal);
				ELSIF stDoneFlags.bSetup THEN
					(* setup done, start "normal" running mode *)
					_bTriggerSetup := FALSE;
					_ActiveChange := BACnetProgramRequest_run;
				END_IF
			ELSE
				IF stFailedFlags.bRun OR bCommonError OR (NOT bRelease) THEN
					(* abort *)
					_ProgramState := TO_WORD(BACnetProgramState_halted);
					_ActiveChange := BACnetProgramRequest_ready;
					_ReasonForHalt  := TO_WORD(BACnetProgramError_progerror_internal);
				ELSIF stDoneFlags.bRun THEN
					(* switch to running state *)
					_ProgramState  := TO_WORD(BACnetProgramState_running);
					_ActiveChange := BACnetProgramRequest_ready;
				END_IF
			END_IF

		BACnetProgramRequest_halt:
			(* wait on halted *)
			IF stFailedFlags.bHalt OR bCommonError OR (NOT bRelease) THEN
				(* abort *)
				_ProgramState := TO_WORD(BACnetProgramState_halted);
				_ActiveChange := BACnetProgramRequest_ready;
				_ReasonForHalt  := TO_WORD(BACnetProgramError_progerror_internal);
			ELSIF stDoneFlags.bHalt THEN
				(* halted *)
				_ProgramState := TO_WORD(BACnetProgramState_halted);
				_ActiveChange := BACnetProgramRequest_ready;
				_ReasonForHalt  := TO_WORD(BACnetProgramError_program);
			END_IF

		BACnetProgramRequest_unload:
			_ProgramState	 := TO_WORD(BACnetProgramState_unloading);
			_ActiveChange	:= BACnetProgramRequest_ready;

	END_CASE

	(* start change request and handle error states *)
	IF (_ActiveChange = BACnetProgramRequest_ready) THEN

		CASE TO_DINT(_ProgramState) OF
			BACnetProgramState_idle:
				IF bCommonError THEN
					(* abort *)
					_ProgramState := TO_WORD(BACnetProgramState_halted);
					_ReasonForHalt  := TO_WORD(BACnetProgramError_progerror_internal);
				ELSIF (NOT bRelease) THEN
					(* abort *)
					_ProgramState := TO_WORD(BACnetProgramState_halted);
					_ReasonForHalt  := TO_WORD(BACnetProgramError_other);
				ELSIF (NOT _bLockedForChange) THEN
					_ReasonForHalt  := TO_WORD(BACnetProgramError_program_normal);
					CASE TO_DINT(_ProgramChange) OF
						BACnetProgramRequest_unload,
						BACnetProgramRequest_halt:
							(* acknowledge without execution *)
							_SetProgramReadyState	:= TRUE;
						BACnetProgramRequest_restart,
						BACnetProgramRequest_run,
						BACnetProgramRequest_load:
							(* execute request *)
							_ActiveChange := BACnetProgramRequest_load;
							_bTriggerSetup := TRUE;
					END_CASE
				END_IF

			BACnetProgramState_loading:
				IF bCommonError THEN
					(* abort *)
					_ProgramState := TO_WORD(BACnetProgramState_halted);
					_ReasonForHalt  := TO_WORD(BACnetProgramError_progerror_internal);
				ELSIF (NOT bRelease) THEN
					(* abort *)
					_ProgramState := TO_WORD(BACnetProgramState_halted);
					_ReasonForHalt  := TO_WORD(BACnetProgramError_other);
				ELSIF stFailedFlags.bLoad THEN
					(* abort *)
					_ProgramState := TO_WORD(BACnetProgramState_halted);
					_ReasonForHalt  := TO_WORD(BACnetProgramError_load_failed);
				ELSIF stDoneFlags.bLoad THEN
					(* DONE *)
					_bTriggerSetup := TRUE;
					_ActiveChange := BACnetProgramRequest_run;
				ELSIF (NOT _bLockedForChange) THEN
					_ReasonForHalt  := TO_WORD(BACnetProgramError_program_normal);
					CASE to_dint(_ProgramChange) OF
						BACnetProgramRequest_load,
						BACnetProgramRequest_run,
						BACnetProgramRequest_halt,
						BACnetProgramRequest_restart:
							(* acknowledge without execution *)
							_SetProgramReadyState	:= TRUE;
						BACnetProgramRequest_unload:
							(* execute request *)
							_ActiveChange := to_int(_ProgramChange);
					END_CASE
				END_IF

			BACnetProgramState_running:
				IF bCommonError THEN
					(* abort *)
					_ProgramState := TO_WORD(BACnetProgramState_halted);
					_ReasonForHalt  := TO_WORD(BACnetProgramError_progerror_internal);
				ELSIF (NOT bRelease) THEN
					(* abort *)
					_ProgramState := TO_WORD(BACnetProgramState_halted);
					_ReasonForHalt  := TO_WORD(BACnetProgramError_other);
				ELSIF bWaitForSomething THEN
					(* wait on something *)
					_ProgramState  := TO_WORD(BACnetProgramState_waiting);
				ELSIF (NOT _bLockedForChange) THEN
					_ReasonForHalt  := TO_WORD(BACnetProgramError_program_normal);
					CASE to_dint(_ProgramChange) OF
						BACnetProgramRequest_run:
							(* is already running *)
							_SetProgramReadyState	:= TRUE;
						BACnetProgramRequest_unload,
						BACnetProgramRequest_halt:
							(* execute request *)
							_ActiveChange := to_int(_ProgramChange);
						BACnetProgramRequest_restart,
						BACnetProgramRequest_load:
							(* retrigger setup *)
							_ActiveChange := BACnetProgramRequest_restart;
							_bTriggerSetup := TRUE;
					END_CASE
				END_IF

			BACnetProgramState_waiting:
				IF bCommonError THEN
					(* abort *)
					_ProgramState := TO_WORD(BACnetProgramState_halted);
					_ReasonForHalt  := TO_WORD(BACnetProgramError_progerror_internal);
				ELSIF (NOT bRelease) THEN
					(* abort *)
					_ProgramState := TO_WORD(BACnetProgramState_halted);
					_ReasonForHalt  := TO_WORD(BACnetProgramError_other);
				ELSIF (NOT bWaitForSomething) THEN
					(* got it *)
					_ProgramState  := TO_WORD(BACnetProgramState_running);
				ELSIF (NOT _bLockedForChange) THEN
					_ReasonForHalt  := TO_WORD(BACnetProgramError_program_normal);
					CASE to_dint(_ProgramChange) OF
						BACnetProgramRequest_run:
							(* is already running *)
							_SetProgramReadyState	:= TRUE;
						BACnetProgramRequest_unload,
						BACnetProgramRequest_halt:
							(* execute request *)
							_ActiveChange := to_int(_ProgramChange);
					END_CASE
				END_IF

			BACnetProgramState_halted:
				IF (NOT bCommonError) AND bRelease AND (NOT _bLockedForChange) THEN
					CASE TO_DINT(_ProgramChange) OF
						BACnetProgramRequest_halt:
							(* acknowledge without execution *)
							_SetProgramReadyState	:= TRUE;
						BACnetProgramRequest_unload:
							(* execute request *)
							_ActiveChange := TO_INT(_ProgramChange);
						BACnetProgramRequest_restart,
						BACnetProgramRequest_load:
							(* retrigger setup *)
							_ActiveChange := BACnetProgramRequest_restart;
							_bTriggerSetup := TRUE;
						BACnetProgramRequest_run:
							(* start, but don't trigger setup *)
							_ActiveChange := TO_INT(_ProgramChange);
							_bTriggerSetup := FALSE;
					END_CASE
				END_IF

			BACnetProgramState_unloading:
				IF bModeUnloadComplex THEN
					_ReasonForHalt  := TO_WORD(BACnetProgramError_program_normal);
					IF bCommonError THEN
						(* abort *)
						_ProgramState := TO_WORD(BACnetProgramState_halted);
						_ActiveChange := BACnetProgramRequest_ready;
						_ReasonForHalt  := TO_WORD(BACnetProgramError_progerror_internal);
					ELSIF (NOT bRelease) THEN
						(* abort *)
						_ProgramState := TO_WORD(BACnetProgramState_halted);
						_ActiveChange := BACnetProgramRequest_ready;
						_ReasonForHalt  := TO_WORD(BACnetProgramError_other);
					ELSIF stFailedFlags.bUnload THEN
						(* abort *)
						_ProgramState := TO_WORD(BACnetProgramState_halted);
						_ActiveChange := BACnetProgramRequest_ready;
						_ReasonForHalt  := TO_WORD(BACnetProgramError_other);
					ELSIF stDoneFlags.bUnload THEN
						(* DONE *)
						_ActiveChange := BACnetProgramRequest_ready;
						_ProgramState  := TO_WORD(BACnetProgramState_idle);
					ELSIF (NOT _bLockedForChange) THEN
						CASE TO_DINT(_ProgramChange) OF
							BACnetProgramRequest_load,
							BACnetProgramRequest_run,
							BACnetProgramRequest_halt,
							BACnetProgramRequest_restart,
							BACnetProgramRequest_unload:
								(* acknowledge without execution *)
								_SetProgramReadyState	:= TRUE;
						END_CASE
					END_IF
				END_IF

		END_CASE
	END_IF

	(* check state of "change" request *)
	IF (_ActiveChange <> BACnetProgramRequest_ready) THEN
		(* request is active, lock execution *)
		_bLockedForChange		:= TRUE;
	ELSIF _bLockedForChange AND (NOT _SetProgramReadyState) THEN
		(* change finished, tell the stack done *)
		_SetProgramReadyState	:= TRUE;
		_bTriggerSetup			:= FALSE;
	ELSIF (TO_INT(_ProgramChange) = BACnetProgramRequest_ready) THEN
		(* wait on new requests *)
		_SetProgramReadyState	:= FALSE;
		_bLockedForChange		:= FALSE;
		_bTriggerSetup			:= FALSE;
	ELSE
		(* new request *)
		_bTriggerSetup			:= FALSE;
	END_IF

	(* external requests *)
	stRequestFlags.bLoad			:= _ProgramState = TO_WORD(BACnetProgramState_loading) AND (NOT _bLockedForChange);
	stRequestFlags.bSetup			:=	(		(_ActiveChange = BACnetProgramRequest_run)
										OR	(_ActiveChange = BACnetProgramRequest_restart)
									)
								AND	_bTriggerSetup;
	stRequestFlags.bRun			:= (_ActiveChange = BACnetProgramRequest_run) AND (NOT _bTriggerSetup);
	stRequestFlags.bHalt			:= _ActiveChange = BACnetProgramRequest_halt;
	stRequestFlags.bUnload		:=	(_ActiveChange = BACnetProgramRequest_unload)
								OR	(		_ProgramState = TO_WORD(BACnetProgramState_unloading)
										AND	(NOT _bLockedForChange)
									);

	(* active status flags *)
	stActiveStateFlags.bIdle		:= _ProgramState = TO_WORD(BACnetProgramState_idle);
	stActiveStateFlags.bLoading		:= _ProgramState = TO_WORD(BACnetProgramState_loading);
	stActiveStateFlags.bRunning		:= _ProgramState = TO_WORD(BACnetProgramState_running);
	stActiveStateFlags.bWaiting		:= _ProgramState = TO_WORD(BACnetProgramState_waiting);
	stActiveStateFlags.bHalted		:= _ProgramState = TO_WORD(BACnetProgramState_halted);
	stActiveStateFlags.bUnloading	:= _ProgramState = TO_WORD(BACnetProgramState_unloading);
ELSE
	(* server device not ready, reset local ready also *)
	bReady := FALSE;
	nErrorId := BACnet_ERR_OPERATIONAL;
END_IF
(* set error flag *)
bError := (nErrorId <> BACnet_ERR_NO_ERROR);

END_FUNCTION_BLOCK

// POUs/BACnet Helper/Flags/F_BACnet_StatusFlags
FUNCTION F_BACnet_StatusFlags : ST_BACnet_StatusFlags
VAR_INPUT
	data	: WORD;
END_VAR
VAR
END_VAR

F_BACnet_StatusFlags.in_alarm:= _F_BACnet_IsBitFieldBitSet( data:=data, bitNbr:=BACnetStatusFlags_in_alarm);
F_BACnet_StatusFlags.fault:= _F_BACnet_IsBitFieldBitSet( data:=data, bitNbr:=BACnetStatusFlags_fault);
F_BACnet_StatusFlags.overridden:= _F_BACnet_IsBitFieldBitSet( data:=data, bitNbr:=BACnetStatusFlags_overridden);
F_BACnet_StatusFlags.out_of_service:= _F_BACnet_IsBitFieldBitSet( data:=data, bitNbr:=BACnetStatusFlags_out_of_service);

END_FUNCTION

// POUs/BACnet Helper/[internal]/_F_BACnet_IsBitFieldBitSet
FUNCTION _F_BACnet_IsBitFieldBitSet : BOOL
VAR_INPUT
	data	:	DWORD;
	bitNbr		:	INT;
END_VAR
VAR
END_VAR

_F_BACnet_IsBitFieldBitSet:= (data AND (SHR(DWORD#16#00008000,_F_BACnet_BitFieldBit(bitNbr)))) > 0;

END_FUNCTION

// POUs/BACnet Helper/[internal]/_F_BACnet_BitFieldBit
FUNCTION _F_BACnet_BitFieldBit : WORD
VAR_INPUT
	bitNbr	:	INT;
END_VAR
VAR
END_VAR

_F_BACnet_BitFieldBit := to_word((bitNbr/8) * 8 + (bitNbr MOD 8));

END_FUNCTION

// POUs/BACnet ADS/[obsolete]/FB_BACnet_NotificationSinkDelEntry
FUNCTION_BLOCK FB_BACnet_NotificationSinkDelEntry
VAR_INPUT
	bExecute	: BOOL;
	nIndex		: UDINT;
	sNetId		: T_AmsNetId;
	nPort		: T_AmsPort;
	tTimeout	: TIME := BACnet_ADSTimeOut;
END_VAR
VAR_OUTPUT
	bBusy		: BOOL;
	bEmpty		: BOOL;
	bError		: BOOL;
	nErrorId	: UDINT;
END_VAR
VAR
	_AdsReadClient	: ADSREAD;
END_VAR

	_AdsReadClient(
		NETID	:= sNetId,
		PORT	:= nPort,
		IDXGRP	:= 16#5,
		IDXOFFS	:= nIndex,
		LEN		:= 0,
		DESTADDR:= 0,
		READ	:= bExecute,
		TMOUT	:= tTimeout,
		BUSY	=> bBusy,
		ERR		=> bError,
		ERRID	=> nErrorId);

	bEmpty := ((UDINT_TO_DWORD(_AdsReadClient.ERRID) AND 16#FFF) = 16#703);

END_FUNCTION_BLOCK

// POUs/BACnet Objects/Remote (Client)/FB_BACnet_RemoteDevice
FUNCTION_BLOCK FB_BACnet_RemoteDevice
VAR_INPUT
	bReset				: BOOL;
	bAutoReset			: BOOL;
	bDisableWOC			: BOOL;
	bReSubscribeCOV		: BOOL;
	bAutoReSubscribe	: BOOL;
	bTriggerWOC			: BOOL; (* Revision 9 feature: FALSE --> TRUE writes all output process data to remote device *)
	bReload				: BOOL; (* Reload ADS connection and increase reload counter (trigger autoget) *)
	nAmsPort			: UINT := 0; (* Optional setting: Ads port of BACnet client, default = not set *)
END_VAR
VAR_OUTPUT
	stAdsConn			: ST_BACnet_AdsConnection;
	eSystemStatus		: E_BACNETDEVICESTATUS;
	bEthLinkOk			: BOOL;
	bGatewayOk			: BOOL;
	sAmsNetId			: T_AmsNetId;
	bEnabledWOC			: BOOL;
	bWOCTriggered		: BOOL;
	bOperational		: BOOL;
	bConnecting			: BOOL;
	bFirstCycle			: BOOL;
	bError				: BOOL;
	nErrorId			: UINT;
	bClientTimeout		: BOOL;
	bServiceFailed		: BOOL;
	nTimeoutCnt			: UDINT;
	nServiceFailCnt		: UDINT;
END_VAR
VAR
	_ObjectId AT%I*:DWORD;			(* ~(BACnet_ObjectIdentifier			:		: LINK ) *)
	_SystemStatus AT%I*	: E_BACNETDEVICESTATUS;	(* ~
										(BACnet_SystemStatus 				: 		: )
										(BACnet_ObjectType					: DEV	: )
										(BACnet_RemoteCycletimeRead 		: 5000	: ) polling each 5 seconds
										(BACnet_RemoteFlagsRead        		: 2     : ) 2 = polling, so the object detects if the client is unreachable!
										(BACnet_RemoteResubscriptionInterval: 240 	: )
										(BACnet_RemoteCycleTimeWrite   		: 1000	: )
										(BACnet_RemoteFlagsWrite       		: 1		: ) *)
	_ClientStatus AT%I*:WORD;		(* ~(BACnet_ClientStatus				:		: )	*)
	_ClientControl AT%Q*:WORD;		(* ~(BACnet_ClientControl				:		: ) *)
	_rtrigReset			: R_TRIG;
	_rtrigOperational	: R_TRIG;
	_rtrigResubscribe	: R_TRIG;
	_rtrigTimeoutCnt	: R_TRIG;
	_rtrigServiceFailCnt: R_TRIG;
	_bReqResubscribe	: BOOL;
	_bComplete			: BOOL;
	_tofTimeoutLeft		: TOF;
	_tofServiceErrLeft	: TOF;
	_ftrigTimeoutLeft	: F_TRIG;

	_bHasStarted		: BOOL := TRUE;
	_nUpdateCount		: UDINT := 0;
	_nUpdateCountAdp 	: UDINT := 0;
	_BACnetAdapter		: POINTER TO FB_BACnet_Adapter;
	_AdsConn			: _FB_BACnet_AdsConn;
	_rtrigReload		: R_TRIG;
	_bLegacyMode		: BOOL;
	_tonAdsReset		: TON;

	_rtrigWOC			: R_TRIG;
	_bTriggerWOC		: BOOL;
	_tonWOCTrigger		: TON;
END_VAR

(* check pointer to bacnet adapter instance *)
IF pBACnet_Adapter > 0 THEN
	_BACnetAdapter := pBACnet_Adapter;
ELSE
	_BACnetAdapter := ADR(fbBACnet_Adapter);
END_IF

(* update server device *)
IF _BACnetAdapter^._nUpdateCount = _nUpdateCountAdp THEN
	_BACnetAdapter^();
END_IF
(* remind current number of update counter *)
_nUpdateCountAdp := _BACnetAdapter^._nUpdateCount;

(* check for client errors *)
_rtrigTimeoutCnt(CLK:= _ClientStatus.0, Q=> );
IF _rtrigTimeoutCnt.Q AND _bComplete THEN
	nErrorId := BACnet_ERR_CLIENT_TIMEOUT;
ELSIF (NOT _ClientStatus.0) THEN
	(* reset acknowledge flag *)
	_ClientControl.0 := FALSE;
END_IF
_rtrigServiceFailCnt(CLK:= _ClientStatus.1, Q=> );
IF _rtrigServiceFailCnt.Q AND _bComplete THEN
	nErrorId := BACnet_ERR_CLIENT_SERVICE;
ELSIF (NOT _ClientStatus.1) THEN
	(* reset acknowledge flag *)
	_ClientControl.1 := FALSE;
END_IF

(* convert SystemStatus to enumeration *)
eSystemStatus := _SystemStatus;
(* reset trigger *)
_rtrigReset(CLK:= bReset, Q=> );
(* reset error ID and flag *)
IF (nErrorId < 20) OR _rtrigReset.Q OR bAutoReset THEN
	nErrorId := BACnet_ERR_NO_ERROR;
END_IF
IF _rtrigReset.Q OR (NOT _bComplete) OR bAutoReset THEN
	_ClientControl.0 := _ClientStatus.0;
	_ClientControl.1 := _ClientStatus.1;
END_IF

(* read NetId and convert to string *)
sAmsNetId := _BACnetAdapter^.sAmsNetId;
(* check if it plausible *)
IF sAmsNetId = '' THEN
	(* NetId not OK, return with error *)
	nErrorId := BACnet_ERR_NO_VALID_NET_ID;
ELSIF (NOT _BACnetAdapter^.bEthLinkOk) THEN
	(* ethernet link missing *)
	nErrorId := BACnet_ERR_NO_ETH_LINK;
ELSIF (NOT _BACnetAdapter^.bGatewayOk) THEN
	(* gateway missing *)
	nErrorId := BACnet_ERR_NO_GATEWAY;
END_IF

(* summerize timeout errors *)
_tofTimeoutLeft(
	IN:= (_rtrigTimeoutCnt.Q AND _bComplete),
	PT:= T#20s,
	Q=> bClientTimeout,
	ET=> );
IF _tofTimeoutLeft.IN THEN
	nTimeoutCnt := nTimeoutCnt + 1;
END_IF
_ftrigTimeoutLeft(CLK:= _tofTimeoutLeft.Q, Q=> );

(* summerize service errors *)
_tofServiceErrLeft(
	IN:= (_rtrigServiceFailCnt.Q AND _bComplete),
	PT:= T#20s,
	Q=> bServiceFailed,
	ET=> );
IF _tofServiceErrLeft.IN THEN
	nServiceFailCnt := nServiceFailCnt + 1;
END_IF

(* WOC trigger control *)
_rtrigWOC(CLK:= bTriggerWOC, Q=> );
IF (_ClientStatus.2 OR bDisableWOC) AND bTriggerWOC THEN
	nErrorId := BACnet_ERR_WOC_DISABLED;
	_bTriggerWOC := FALSE;
ELSIF _ClientStatus.4 OR _bTriggerWOC THEN
	IF _rtrigWOC.Q THEN
		nErrorId := BACnet_ERR_WOC_TRIGGER_ACTIVE;
	ELSIF (NOT bTriggerWOC) THEN
		_bTriggerWOC := FALSE;
	END_IF
ELSIF _rtrigWOC.Q THEN
	_bTriggerWOC := TRUE;
END_IF

(* controls *)
_ClientControl.2 := bDisableWOC;
_ClientControl.3 := _bReqResubscribe;
_ClientControl.4 := _bTriggerWOC;
_ClientControl.5 := (NOT _bHasStarted); (* a-life flag *)

(* states *)
bEthLinkOk := _BACnetAdapter^.bEthLinkOk;
bGatewayOk := _BACnetAdapter^.bGatewayOk;

bEnabledWOC := (NOT _ClientStatus.2);
bConnecting := (SHR((_ClientStatus AND 16#FF00), 8) < 4);
_bComplete :=		(NOT bConnecting)
				AND	(_SystemStatus = 0)
				AND	_BACnetAdapter^.bEthLinkOk;
bOperational :=		_bComplete
				AND ((NOT _ClientStatus.0) OR bAutoReset);
bWOCTriggered	:= bTriggerWOC AND _ClientStatus.4 AND (NOT (_ClientStatus.2 OR bDisableWOC));

(* Resubscribe COV *)
_rtrigOperational(CLK:= bOperational, Q=> );
_rtrigResubscribe(CLK:= bReSubscribeCOV, Q=> );
IF		(		(		(		_rtrigOperational.Q
							OR (_ftrigTimeoutLeft.Q AND bAutoReset)
						)
					AND	bAutoReSubscribe
				)
			OR	_rtrigResubscribe.Q
		)
	AND	(NOT _bReqResubscribe)
THEN
	(* operation mode reached or resubscription was externally triggered, start resubcription *)
	_bReqResubscribe	:= TRUE;
ELSIF (NOT bOperational) THEN
	(* not operational *)
	_bReqResubscribe	:= FALSE;
ELSE
	IF _bReqResubscribe AND _ClientStatus.3 THEN
		(* resubscription triggered *)
		_bReqResubscribe := FALSE;
	END_IF
END_IF

(* check WOC trigger state *)
_tonWOCTrigger(IN:= _bTriggerWOC, PT:= T#5s, Q=> , ET=> );
IF _tonWOCTrigger.Q THEN
	nErrorId := BACnet_ERR_WOC_TRIGGER_UNSUP;
	IF (NOT bTriggerWOC) THEN
		_bTriggerWOC := FALSE;
	END_IF
END_IF

(* reload ADS connection *)
_rtrigReload(CLK:= bReload, Q=> );
IF _rtrigReload.Q AND (NOT _AdsConn.bBusy) THEN
	_bLegacyMode := FALSE;
	_AdsConn(
		bAutoReload		:= FALSE,
		bReload			:= FALSE,
		bDevOperational	:= bOperational,
		sAmsNetId		:= sAmsNetId,
		tDevObjId		:= _ObjectId);
END_IF
(* probe ADS connection parameter *)
IF (NOT _bLegacyMode) AND _bComplete AND (_ObjectId <> 0) THEN
	(* call ADS connection *)
	_AdsConn(
		bAutoReload		:= TRUE,
		bReload			:=	(bReset AND (NOT _AdsConn.bReady) AND (NOT bAutoReset))
						OR	_tonAdsReset.Q
						OR	_ftrigTimeoutLeft.Q
						OR	bReload,
		bIsClient		:= TRUE,
		bDevOperational	:= bOperational,
		sAmsNetId		:= sAmsNetId,
		tDevObjId		:= _ObjectId,
		bReady			=> ,
		bBusy			=> ,
		bDone			=> ,
		bError			=> ,
		nErrorId		=> ,
		stBACnetAds		=> stAdsConn);

	(* error when ADS connection failed *)
	IF _AdsConn.bError THEN
		IF (_AdsConn.nErrorId = BACnet_ERR_ADS_LegacyStack) THEN
			_bLegacyMode := TRUE;
			stAdsConn.nReload := stAdsConn.nReload + 1;
		ELSIF (nErrorId = 0) THEN
			nErrorId := _AdsConn.nErrorId;
		END_IF
	END_IF

	(* auto reload when error is active *)
	_tonAdsReset(
		IN:=	(NOT _AdsConn.bReload)
			AND	_AdsConn.bError
			AND	bAutoReset
			AND bOperational,
		PT:= t#2s,
		Q=> ,
		ET=> );
END_IF
IF _bLegacyMode THEN
	stAdsConn.bClient	:= TRUE;
	stAdsConn.bServer	:= FALSE;
	stAdsConn.bValid	:= (nAmsPort >= 1000);
	stAdsConn.nAmsPort	:= nAmsPort;
	stAdsConn.sAmsNetId	:= sAmsNetId;
	stAdsConn.nDeviceId	:= F_BACnet_GetObjInstance(_ObjectId);
END_IF


bError := (nErrorId <> BACnet_ERR_NO_ERROR);

(* update counter *)
IF (_nUpdateCount = 0) AND _bHasStarted THEN
	bFirstCycle := TRUE;
	_bHasStarted := FALSE;
ELSE
	bFirstCycle := FALSE;
END_IF
_nUpdateCount := _nUpdateCount + 1;

END_FUNCTION_BLOCK

// POUs/BACnet Objects/Local (Server)/FB_BACnet_Loop
FUNCTION_BLOCK FB_BACnet_Loop
VAR_INPUT
	fAccLimit		: REAL := 0.0; (* Setpoint acceleration limit positive and negative [1/s] *)
END_VAR
VAR_IN_OUT
	Device			: FB_BACnet_Device;
END_VAR
VAR_OUTPUT
	bReady			: BOOL;
	fSetPoint		: REAL;
	fControlledValue: REAL;
	fPresentValue	: REAL;
	fPropBand		: REAL; (* controller output in range of -100...100% in relation to Min.-/Max.-output *)
	bOverridden		: BOOL;
	bOutOfService	: BOOL;
	bFault			: BOOL;
	bInAlarm		: BOOL;
	bOpenLoop		: BOOL;
	bCommFailure	: BOOL;
	bOtherFault		: BOOL;
	bError			: BOOL;
	nErrorId		: UINT;
	eMode			: E_BACNETLOOPMODE; (* mode is detected by the unit of property Integral_Constant and Derivative_Constant (Time_seconds = BACnetLoopMode_Standard) *)
END_VAR
VAR
	_ControlledVariableValue AT%I*: REAL;	(* ~(BACnet_ControlledVariableValue :		: )
												(BACnet_ObjectType				: LOOP	: )	*)
	_Setpoint AT%I*:REAL;					(* ~(BACnet_Setpoint				:		: )	*)
	_ProportionalConstant AT%I*:REAL;		(* ~(BACnet_ProportionalConstant	:		: )	*)
	_IntegralConstant AT%I*:REAL;			(* ~(BACnet_IntegralConstant	 	:		: )	*)
	_DerivativeConstant AT%I*:REAL;			(* ~(BACnet_DerivativeConstant	 	:		: )	*)
	_MaximumOutput AT%I*:REAL;				(* ~(BACnet_MaximumOutput			:		: )	*)
	_MinimumOutput AT%I*:REAL;				(* ~(BACnet_MinimumOutput			:		: )	*)
	_Bias AT%I*:REAL;						(* ~(BACnet_Bias					:		: )	*)
	_PresentValueI AT%I*: REAL; 			(* ~(BACnet_PresentValue 			: 		: )	*)
	_StatusFlags AT%I*: WORD; 				(* ~(BACnet_StatusFlags 			: 		: )	*)
	_Reliability AT%I*: WORD;(* ~(BACNET_RELIABILITY 			:		: )	*)
	_ControlAction AT%I*:E_BACNETACTION;	(* ~(BACNET_ACTION				 	:		: )	*)
	_PropConstantUnits AT%I*:E_BACNETUNIT;	(* ~(BACnet_ProportionalConstantUnits:	Other_no_units	: WRITEPROTECT) *)
	_IntegralConstUnits AT%I*:E_BACNETUNIT;	(* ~(BACnet_IntegralConstantUnits	:	Other_no_units	: WRITEPROTECT) *)
	_DerivativeConstUnits AT%I*:E_BACNETUNIT;(*~(BACnet_DerivativeConstantUnits	:	Other_no_units	: WRITEPROTECT) *)
	_PresentValueQ AT%Q*: REAL;				(* ~(BACnet_PresentValue	 		:		: )	*)
	_StatusFlagsBits : ST_BACnet_StatusFlags;

	_sysTime	: GETCPUCOUNTER;
	_Time		: T_LARGE_INTEGER;
	_TimeOld	: T_LARGE_INTEGER;
	_cycleTime	: REAL;
	_PidControl : FB_BACnet_PidControl;
	_fbAccLimit : FB_BACnet_AccLimit;

	_nUpdateCount : UDINT := 0;
END_VAR

(* update server device *)
IF (Device._nUpdateCount = _nUpdateCount) THEN
	Device();
END_IF
(* remind current number of update counter *)
_nUpdateCount := Device._nUpdateCount;

(* determine cycle time *)
_TimeOld := _Time;
_sysTime(cpuCntLoDW=> _Time.dwLowPart, cpuCntHiDW=> _Time.dwHighPart);
_cycleTime := _F_BACnet_SysTimeDiff(In1:=_Time, In2:=_TimeOld);

(* check BitString format of StatusFlags --> if StatusFlags are less than 4, object isn't linked correctly *)
IF (_StatusFlags < 4) THEN
	(* wrong mapping *)
	nErrorId := BACnet_ERR_WRONG_MAPPING;
	bReady := FALSE;

ELSIF Device.bOperational THEN
	(* ready state *)
	bReady := TRUE;
	nErrorId := BACnet_ERR_NO_ERROR;

	(* decode status flags *)
	_StatusFlagsBits := F_BACnet_StatusFlags(_StatusFlags);

	(* copy states to output *)
	bOverridden := _StatusFlagsBits.overridden;
	bOutOfService := _StatusFlagsBits.out_of_service;
	bFault := _StatusFlagsBits.fault;
	bInAlarm := _StatusFlagsBits.in_alarm;
	bOpenLoop := (_Reliability = TO_WORD(BACnetReliability_open_loop));
	bCommFailure := (_Reliability = TO_WORD(BACnetReliability_communication_failure));
	bOtherFault := (_Reliability = TO_WORD(BACnetReliability_unreliable_other));

	(* check PID mode *)
	IF		((_IntegralConstUnits = BACnetUnit_Time_seconds OR _IntegralConstUnits = 0) AND _DerivativeConstUnits = BACnetUnit_Time_seconds)
		AND	((_DerivativeConstUnits = BACnetUnit_Time_seconds OR _DerivativeConstUnits = 0) AND _IntegralConstUnits = BACnetUnit_Time_seconds)
		AND (_PropConstantUnits = BACnetUnit_Other_no_units)
	THEN
		(* both are time_seconds *)
		eMode := BACnetLoopMode_Standard;
	ELSIF	(_IntegralConstUnits <> BACnetUnit_Time_seconds)
		AND	(_DerivativeConstUnits <> BACnetUnit_Time_seconds)
		AND (_PropConstantUnits = BACnetUnit_Other_no_units)
		(* both are not time_seconds *)
	THEN
		eMode := BACnetLoopMode_Ideal;
	ELSE
		(* unknown settings - stop controller *)
		eMode := BACnetLoopMode_None;
	END_IF

	(* check reliability and mode *)
	IF		_Reliability <> to_word(BACnetReliability_no_fault_detected)
		OR	(eMode = BACnetLoopMode_None)
	THEN
		_PidControl.bReset			:= TRUE;

	(* is set out of service? *)
	ELSIF _StatusFlagsBits.out_of_service THEN
		_PidControl.bReset			:= TRUE;

	(* decide the control action (direct or reverse) *)
	ELSIF _ControlAction = BACnetAction_direct THEN
		_PidControl.bReset			:= FALSE;
		_PidControl.fPresentValue	:= _ControlledVariableValue;
		_PidControl.fSetpoint		:= _Setpoint;

	ELSIF _ControlAction = BACnetAction_reverse THEN
		_PidControl.bReset			:= FALSE;
		_PidControl.fPresentValue	:= _Setpoint;
		_PidControl.fSetpoint		:= _ControlledVariableValue;

	ELSE
		(* unknown action *)
		_PidControl.bReset			:= TRUE;
	END_IF

	(* set parameter depending on mode *)
	CASE eMode OF
		BACnetLoopMode_Ideal:
			_PidControl.fKp := _ProportionalConstant;
			_PidControl.fKi	:= _IntegralConstant;
			_PidControl.fKd	:= _DerivativeConstant;
		BACnetLoopMode_Standard:
			(* Kp = Kp *)
			_PidControl.fKp := _ProportionalConstant;
			(* Ki = Kp / Ti *)
			IF (_IntegralConstant <> 0.0) THEN
				_PidControl.fKi	:= _ProportionalConstant / _IntegralConstant;
			ELSE
				_PidControl.fKi	:= 0.0;
			END_IF
			(* Kd = Kp * Td *)
			_PidControl.fKd	:= _ProportionalConstant * _DerivativeConstant;
	END_CASE

	(* call PID control function block *)
	_PidControl(
		fCtrlCycleTime	:= _cycleTime,
		fBias			:= _Bias,
		fTp				:= -1.0,
		fMaxOutput		:= _MaximumOutput,
		fMinOutput		:= _MinimumOutput,
		nErrorStatus	=>
	);
	_fbAccLimit.X := _PidControl.fY;

	(* set other outputs *)
	fSetPoint := _Setpoint;
	fPresentValue := _PresentValueI;
	fControlledValue := _ControlledVariableValue;
ELSE
	(* server device not ready, reset local ready also *)
	bReady := FALSE;
	nErrorId := BACnet_ERR_OPERATIONAL;
END_IF

(* limit present value *)
_fbAccLimit(X:= , Amax:= fAccLimit, Tcycle:= _cycleTime, Y=> _PresentValueQ, A=> );

(* calculate proportional band *)
IF (_MaximumOutput > 0.0) AND (_MinimumOutput >= 0.0) THEN
	fPropBand := ((_PresentValueQ - _MinimumOutput) / (_MaximumOutput - _MinimumOutput)) * 100.0;
ELSIF (_MaximumOutput <= 0.0) AND (_MinimumOutput < 0.0) THEN
	fPropBand := ((_PresentValueQ - _MaximumOutput) / (_MaximumOutput - _MinimumOutput)) * 100.0;
ELSIF (_PresentValueQ > 0.0) AND (_MaximumOutput > 0.0) THEN
	fPropBand := (_PresentValueQ / _MaximumOutput) * 100.0;
ELSIF (_PresentValueQ < 0.0) AND (_MinimumOutput < 0.0) THEN
	fPropBand := (_PresentValueQ / _MinimumOutput) * -100.0;
ELSE
	fPropBand := 0.0;
END_IF

(* set error flag *)
bError := (nErrorId <> BACnet_ERR_NO_ERROR);

END_FUNCTION_BLOCK

// POUs/BACnet Helper/[internal]/_F_BACnet_SysTimeDiff
FUNCTION _F_BACnet_SysTimeDiff : REAL
VAR_INPUT
	In1, In2 : T_LARGE_INTEGER;
END_VAR

_F_BACnet_SysTimeDiff := LREAL_TO_REAL(INT64_TO_LREAL(Int64Sub64(In1, In2)) / 10000000.0); (* [s] *)

END_FUNCTION

// POUs/BACnet Helper/FB_BACnet_PidControl
FUNCTION_BLOCK FB_BACnet_PidControl
VAR_INPUT
	(* controller input  *)
	fSetpoint				: REAL;	(* setpoint value *)
	fPresentValue			: REAL;	(* actual value *)
	(* reset flag *)
	bReset					: BOOL;
	(* controller values *)
	fCtrlCycleTime			: REAL; (* controller cycle time in seconds [s] *)

	fBias					: REAL; (* bias also active when reset is set to 1 *)
	fKp						: REAL;	(* proportional gain Kp	(P) *)
	fKi						: REAL; (* integral gain Ki (I) *)
	fKd						: REAL;	(* derivative gain Kd (D) *)
	fTp						: REAL := -1.0;	(* damping time Tp (PT1) [s] (fTp < 0 --> Tp = Kd / 10) *)

	(* maximum ratings *)
	fMaxOutput				: REAL;
	fMinOutput				: REAL;
END_VAR
VAR_OUTPUT
	fY						: REAL; (* controller output command *)
	nErrorStatus			: UINT; (* controller error output (0: no error; >0:error) *)
END_VAR
VAR
	(* Internal Variable *)
	_fE		: REAL;
	_fEOld	: REAL;
	_fYp	: REAL;
	_fYi	: REAL;
	_fYd	: REAL;
	_fbYd	: FB_BACnet_PT1;
END_VAR

(* preset error number *)
nErrorStatus	:= BACnet_ERR_NO_ERROR;

(* check cycle time parameter: (CycleTime > 0) *)
IF (fCtrlCycleTime <= 0.0) THEN
	nErrorStatus := BACnet_ERR_INVALID_CYCLETIME;
	bReset := TRUE;
END_IF;

(* check controller parameters: (Kp, Ki, Kd >= 0) *)
IF ((fKp < 0.0) OR (fKi < 0.0) OR (fKd < 0.0)) THEN
	nErrorStatus := BACnet_ERR_INVALID_PARAMETER;
	bReset := TRUE;
END_IF;

(* controller reset *)
IF bReset THEN
	(* reset internal and external variables *)
	_fEOld	:= 0.0;
	fY		:= MAX(MIN(fBias, fMaxOutput), fMinOutput);
	_fYi	:= 0.0;
	_fbYd(X:= 0.0, T:= 0.0, Y=> );
	RETURN;
END_IF

(* 3. save old variable *)
_fEOld := _fE;

(* 4. set error/deviation input *)
_fE := fSetpoint - fPresentValue;

(* 5. YP-part *)
_fYp := fKp * _fE;

(* 6. YI-part *)
IF (fKi = 0.0) THEN
	_fYi	:= 0.0;
ELSE
	_fYi := _fYi + (fKi * fCtrlCycleTime * _fE);
END_IF
IF (_fYi > fMaxOutput) THEN
	(* limit wind up positive *)
	_fYi := fMaxOutput;
ELSIF (_fYi < fMinOutput) THEN
	(* limit wind up negative *)
	_fYi := fMinOutput;
END_IF

(* 7. YD-part *)
IF (fTp < 0.0) THEN
	fTp := fKd / 10.0;
END_IF
_fYd := fKd * (_fE - _fEOld) / fCtrlCycleTime;
_fbYd(X:= _fYd, T:= fTp, Tcycle:= fCtrlCycleTime, Y=> );

(* 8. Ysum = YP + YI + YD + Bias and output *)
fY := _fYp + _fYi + _fbYd.Y + fBias;
fY := MAX(MIN(fY, fMaxOutput), fMinOutput);

END_FUNCTION_BLOCK

// POUs/BACnet Helper/FB_BACnet_PT1
FUNCTION_BLOCK FB_BACnet_PT1
VAR_INPUT
	X : REAL; (* input value *)
	T : REAL; (* damping time [s] *)
	Tcycle : REAL; (* cycle time [s] of task; 0 = use internal measuring *)
END_VAR
VAR_OUTPUT
	Y : REAL; (* damped value *)
END_VAR
VAR
	_sysTime	: GETCPUCOUNTER;
	_Time		: T_LARGE_INTEGER;
	_TimeOld	: T_LARGE_INTEGER;
	_cycleTime	: REAL;
	_Yold : REAL;
	_FirstScan : BOOL := TRUE;
END_VAR

(* determine cycle time *)
IF Tcycle = 0.0 THEN
	_TimeOld := _Time;
	_sysTime(cpuCntLoDW=> _Time.dwLowPart, cpuCntHiDW=> _Time.dwHighPart);
	_cycleTime := _F_BACnet_SysTimeDiff(In1:=_Time, In2:=_TimeOld);
ELSE
	_cycleTime := Tcycle;
END_IF

(* exit on wrong cycle time *)
IF _cycleTime <= 0.0 THEN
	RETURN;
END_IF

(* initialize and check on zero/negative damping time *)
IF (T <= 0.0) OR _FirstScan THEN
	Y := X;
	_Yold := Y;
	_FirstScan := FALSE;
	RETURN;
END_IF

(* remind last result *)
_Yold := Y;

(* calculate result *)
Y := 1 / ((T / _cycleTime) + 1) * (X - _Yold) + _Yold;

END_FUNCTION_BLOCK

// POUs/BACnet Helper/FB_BACnet_AccLimit
FUNCTION_BLOCK FB_BACnet_AccLimit
VAR_INPUT
	X : REAL; (* input value [1] *)
	Amax : REAL; (* maximum acceleration of X [1/s]; 0 = limit disabled *)
	Tcycle : REAL; (* cycle time [s] of task; 0 = use internal measuring *)
END_VAR
VAR_OUTPUT
	Y : REAL; (* limited X value [1] *)
	A : REAL; (* input acceleration [1/s] *)
END_VAR
VAR
	_sysTime	: GETCPUCOUNTER;
	_Time		: T_LARGE_INTEGER;
	_TimeOld	: T_LARGE_INTEGER;
	_cycleTime	: REAL;
	_bFirstScan	: BOOL:=TRUE;
	_foldY		: REAL;
END_VAR

(* determine cycle time *)
IF Tcycle = 0.0 THEN
	_TimeOld := _Time;
	_sysTime(cpuCntLoDW=> _Time.dwLowPart, cpuCntHiDW=> _Time.dwHighPart);
	_cycleTime := _F_BACnet_SysTimeDiff(In1:=_Time, In2:=_TimeOld);
ELSE
	_cycleTime := Tcycle;
END_IF

IF (NOT _bFirstScan) THEN
	(* exit on wrong cycle time *)
	IF _cycleTime <= 0.0 THEN
		RETURN;
	END_IF
	(* calculate current acceleration *)
	A := (X - _foldY) / _cycleTime;
	IF (Amax <> 0.0) THEN
		Amax := ABS(Amax);
		IF (ABS(A) > Amax) THEN
			IF (A >= 0.0) THEN
				Y := _foldY + (Amax * _cycleTime);
			ELSE
				Y := _foldY - (Amax * _cycleTime);
			END_IF
		ELSE
			Y := X;
		END_IF
	ELSE
		Y := X;
	END_IF
ELSE
	Y := X;
END_IF

_foldY := Y;
_bFirstScan:=FALSE;

END_FUNCTION_BLOCK

// POUs/BACnet Helper/Real/F_BACnet_RealNull
FUNCTION F_BACnet_RealNull : DWORD
(* function that generates <not-a-number> real state *)

F_BACnet_RealNull:=16#7FFF0000;

END_FUNCTION

// POUs/BACnet Helper/[internal]/F_BACnet_AnalogPV
FUNCTION F_BACnet_AnalogPV : REAL
VAR_INPUT
	bEnable	: BOOL; (* TRUE = commit to stack, FALSE = do-nothing *)
	bNull	: BOOL; (* TRUE = clear priority, FALSE = write value from input *)
	rValue	: REAL;
END_VAR
VAR
	pres : POINTER TO DWORD;
END_VAR

IF (bEnable) THEN
	IF (bNull) THEN
		pres := ADR(F_BACnet_AnalogPV);
		pres^ := F_BACnet_RealNull(); 
	ELSE
		F_BACnet_AnalogPV := rValue;
	END_IF
ELSE
	F_BACnet_AnalogPV := F_BACnet_NAN();
END_IF

END_FUNCTION

// POUs/BACnet Helper/Real/F_BACnet_NAN
FUNCTION F_BACnet_NAN : REAL
(* function that generates <not-a-number> real state *)
VAR
	res : POINTER TO DWORD;
END_VAR

res:=ADR(F_BACnet_NAN);
res^:=16#7FFFFFFF;

END_FUNCTION

// POUs/BACnet Helper/MultiState/F_BACnet_MultiStatePV
FUNCTION F_BACnet_MultiStatePV : UDINT
VAR_INPUT
	bEnable	: BOOL; (* TRUE = commit to stack, FALSE = do-nothing *)
	bNull	: BOOL; (* TRUE = clear priority, FALSE = write number from state input *)
	nState	: UDINT; (* multi-state [1..max-number-of-states] *)
END_VAR

IF (bEnable) THEN
	IF (bNull) THEN
		F_BACnet_MultiStatePV := 16#0;
	ELSE
		F_BACnet_MultiStatePV := nState;
	END_IF
ELSE
	F_BACnet_MultiStatePV := 16#FFFFFFFF;
END_IF

END_FUNCTION

// POUs/BACnet ADS/Properties/FB_BACnet_DescriptionProperty
FUNCTION_BLOCK FB_BACnet_DescriptionProperty
VAR_INPUT
	tObjectID			: T_BACnet_ObjectIdentifier := 16#FFFFFFFF;
	bAutoGet			: BOOL:=TRUE; (* TRUE = get data from property when ADS connection OR object ID changed *)
	bGet				: BOOL; (* FALSE --> TRUE = get data from property *)
END_VAR
VAR_IN_OUT
	stAdsConn			: ST_BACnet_AdsConnection;
END_VAR
VAR_OUTPUT
	bDone				: BOOL;
	bBusy				: BOOL;
	bError				: BOOL;
	nErrorId			: UINT;
	sText				: T_MaxString; (* Object description *)
END_VAR
VAR
	_fbReadProp		: FB_BACnet_ReadProp;
	_i				: INT;
	_rtrigGetSet	: R_TRIG;
	_nAdsReloadOld	: USINT;
	_tObjectIDOld	: T_BACnet_ObjectIdentifier := 16#FFFFFFFF;
	_StringExtDecode: FB_BACnet_StringExtDecode;
END_VAR

(* ADS read *)
_fbReadProp(
	BACnetDevicePort	:= stAdsConn.nAmsPort,
	bExecute			:= ,
	sNetId				:= stAdsConn.sAmsNetId,
	ObjectType			:= F_BACnet_GetObjType(tObjectID),
	PropertyID			:= BACnetPropertyIdentifier_Description,
	DataType			:= BACnetDataType_CharacterStringExt,
	ObjectInstance		:= F_BACnet_GetObjInstance(tObjectID),
	ptrValue			:= ADR(sText),
	nLenValue			:= SIZEOF(sText)-1,
	bDone				=> ,
	bBusy				=> ,
	bError				=> ,
	nErrID				=> ,
	nProcessedLen		=> );

(* trigger start event *)
_rtrigGetSet(CLK:= bGet, Q=> );

(* state machine *)
CASE _i OF

	0: (* Idle *)
		IF		(		(		_rtrigGetSet.Q
							OR	(_nAdsReloadOld <> stAdsConn.nReload)
							OR	(_tObjectIDOld <> tObjectID)
						)
					AND	bAutoGet
				)
			OR	_rtrigGetSet.Q
		THEN
			IF (NOT stAdsConn.bValid) THEN
				(* ADS connection not valid *)
				nErrorId := BACnet_ERR_INVALID_ADS_CONN;
			ELSIF (NOT stAdsConn.bServer AND NOT stAdsConn.bClient) THEN
				(* not a server nor a client *)
				nErrorId := BACnet_ERR_ADS_NoServerClient;
			ELSE
				nErrorId := BACnet_ERR_NO_ERROR;
				_i := 1;
				sText := '';
				(* remind ADS reload counter and parameter *)
				_nAdsReloadOld := stAdsConn.nReload;
				_tObjectIDOld := tObjectID;
			END_IF
			(* reset done flag *)
			bDone := FALSE;
		END_IF
		IF (NOT bGet) AND (NOT bAutoGet) THEN
			nErrorId := BACnet_ERR_NO_ERROR;
			bDone := FALSE;
		END_IF

	(* READ *)
	1: (* read object property data over ADS *)
		IF _fbReadProp.bExecute THEN
			IF _fbReadProp.bError THEN
				_i := 100;
				nErrorId := BACnet_ERR_ADS_Read;
				_fbReadProp.bExecute := FALSE;
			ELSIF (NOT _fbReadProp.bBusy) THEN
				_fbReadProp.bExecute := FALSE;
				(* decode property data *)
				_StringExtDecode(
					pChrStringExt	:= ADR(sText),
					cbOutSize		:= _fbReadProp.nProcessedLen,
					pOutString		:= ADR(sText),
					bValid			=> ,
					bOverflow		=> ,
					nLength			=> ,
					eSrcEncoding	=> );
				(* check overflow flag *)
				IF _StringExtDecode.bOverflow THEN
					nErrorId := BACnet_ERR_ADS_BufferSize;
				ELSIF (NOT _StringExtDecode.bValid) THEN
					nErrorId := BACnet_ERR_ADS_Encoding;
				END_IF
				(* DONE *)
				_i := 100;
			END_IF
		ELSE
			_fbReadProp.bExecute := TRUE;
		END_IF

	100: (* Done *)
		bDone := (nErrorId = BACnet_ERR_NO_ERROR);
		_i := 0;

END_CASE

(* set error flag *)
bError 	:= nErrorId > BACnet_ERR_NO_ERROR;
bBusy 	:= _i > 0;

END_FUNCTION_BLOCK

// POUs/BACnet Helper/String/FB_BACnet_StringExtDecode
FUNCTION_BLOCK FB_BACnet_StringExtDecode (* convert UTF-8/UCS2/UCS4/ISO8859-1 to Windows-1252 *)
VAR_INPUT
	pChrStringExt	: POINTER TO ST_BACnet_CharacterStringExt; (* BACnet character string data structure (header and string) *)
	pOutString		: POINTER TO T_MaxString; (* pointer to result buffer (Windows-1252 encoded) *)
	cbOutSize		: UDINT; (* byte size *)
END_VAR
VAR_OUTPUT
	bValid			: BOOL; (* Decoding successfull *)
	bOverflow		: BOOL; (* String length overflow (source string too long) *)
	bUnsupported	: BOOL; (* Souce encoding is unsupported (use ReadProp function and decode manually instead) *)
	nLength			: UDINT; (* out character length *)
	eSrcEncoding	: E_BACNETSTRINGENCODINGTYPES; (* input encoding *)
END_VAR
VAR
	pText 			: POINTER TO BYTE;
	pByte			: POINTER TO BYTE;
END_VAR

(* preset valid to FALSE *)
bValid := FALSE;
bOverflow := FALSE;
bUnsupported := FALSE;
(* check pointer *)
IF (pChrStringExt = 0) OR (pOutString = 0) THEN
	nLength := 0;
(* check input size *)
ELSIF (cbOutSize = 0) THEN
	(* NULL string *)
	bValid := TRUE;
	pOutString^ := '';
	nLength := 0;
	eSrcEncoding := BACnetStringEncodingTypes_AnsiUtf8;
ELSE
	(* string data available *)
	IF (pChrStringExt^.cookie = 0) THEN
		(* new character string type *)
		nLength			:= UDINT_TO_UINT(pChrStringExt^.strLen);
		eSrcEncoding	:= UDINT_TO_INT(pChrStringExt^.encoding);
		pText			:= ADR(pChrStringExt^.stringData);
	ELSE
		(* ASCII/UTF-8 string *)
		nLength			:= _F_BACnet_ChrStrExtLen(pChrStringExt^);
		eSrcEncoding	:= BACnetStringEncodingTypes_AnsiUtf8;
		pText			:= pChrStringExt;
	END_IF

	(* check size *)
	IF (nLength = 0) THEN
		(* no data *)
		bValid := TRUE;
		pOutString^ := '';
	ELSIF (nLength <= cbOutSize) THEN
		(* copy to output buffer first *)
		MEMMOVE(destAddr:= pOutString, srcAddr:= pText, n:= nLength);

		(* decode and copy *)
		CASE eSrcEncoding OF

			BACnetStringEncodingTypes_AnsiUtf8:
				bValid := TRUE;
				nLength := UDINT_TO_UINT(_F_BACnet_DecodeUTF8(pOutString, nLength));

			BACnetStringEncodingTypes_UCS2:
				bValid := TRUE;
				nLength := UDINT_TO_UINT(_F_BACnet_DecodeUCS2(pOutString, nLength));

			BACnetStringEncodingTypes_UCS4:
				bValid := TRUE;
				nLength := UDINT_TO_UINT(_F_BACnet_DecodeUCS4(pOutString, nLength));

			BACnetStringEncodingTypes_ISO8859:
				bValid := TRUE;
				(* check if string termination is already part of string *)
				pByte := pOutString + nLength - 1;
				IF (pByte^ = 16#00) THEN
					(* termination already part of string *)
					nLength := nLength - 1;
				ELSE
					(* add string termination *)
					pByte := pOutString + nLength;
					pByte^ := 16#00;
				END_IF

			ELSE
				bUnsupported := TRUE;

		END_CASE
	ELSE
		(* text too long *)
		nLength := 0;
		pOutString^ := '';
		bOverflow := TRUE;
	END_IF
END_IF

END_FUNCTION_BLOCK

// POUs/BACnet Helper/[internal]/_F_BACnet_ChrStrExtLen
FUNCTION _F_BACnet_ChrStrExtLen : UDINT

VAR
	pByte	: POINTER TO BYTE;
	nLen	: UDINT;
END_VAR
(*All VAR_IN_OUT variables have been moved to the end of the declaration due to compatibility reasons*)
VAR_IN_OUT
	stCharStringExt	: ST_BACnet_CharacterStringExt;
END_VAR

pByte := ADR(stCharStringExt);
nLen := SIZEOF(stCharStringExt);
(* check the string type *)
IF (nLen > 4 AND stCharStringExt.cookie = 0) THEN
	(* character string ext. *)
	IF (stCharStringExt.strLen <= SIZEOF(stCharStringExt.stringData)) THEN
		(* plausible string length given *)
		_F_BACnet_ChrStrExtLen := stCharStringExt.strLen;
		RETURN;
	END_IF
	(* use sizeof, because string length isn't plausible *)
	nLen := SIZEOF(stCharStringExt.stringData);
	(* re-adjust pointer *)
	pByte := ADR(stCharStringExt.stringData);
END_IF
(* scan zero termination *)
_F_BACnet_ChrStrExtLen := 0;
WHILE ((pByte^ <> 0) AND (_F_BACnet_ChrStrExtLen < nLen)) DO
	pByte := pByte + 1;
	_F_BACnet_ChrStrExtLen := _F_BACnet_ChrStrExtLen + 1;
END_WHILE

END_FUNCTION

// POUs/BACnet Helper/[internal]/_F_BACnet_DecodeUTF8
FUNCTION _F_BACnet_DecodeUTF8 : UDINT (* result is the new character length of the string *)
VAR_INPUT
	pString		: POINTER TO BYTE; (* pointer to UTF-8 string beginning *)
	cbString	: UDINT; (* byte size of string (use SIZEOF - don't use LEN) *)
END_VAR
VAR
	i			: UDINT;
	pResult		: POINTER TO BYTE;
	pBy			: POINTER TO BYTE;
	pByArr		: POINTER TO ARRAY[0..3] OF BYTE;
END_VAR

pResult	:= pString;
pBy		:= pString;
FOR i := 0 TO cbString-1 DO
	pByArr := pBy;
	IF (pByArr^[0] AND 16#F0) = 16#C0 THEN
		IF (pByArr^[1] AND 16#80) = 16#80 THEN
			pResult^ := _F_BACnet_Utf8ToWin1252(pByArr, 2);
			pBy := pBy + 2;
		END_IF
	ELSIF (pByArr^[0] AND 16#F0) = 16#E0 THEN
		IF (pByArr^[1] AND 16#80) = 16#80 THEN
			IF (pByArr^[2] AND 16#80) = 16#80 THEN
				pResult^ := _F_BACnet_Utf8ToWin1252(pByArr, 3);
				pBy := pBy + 3;
			END_IF
		END_IF
	ELSIF (pByArr^[0] AND 16#F0) = 16#F0 THEN
		IF (pByArr^[1] AND 16#80) = 16#80 THEN
			IF (pByArr^[2] AND 16#80) = 16#80 THEN
				IF (pByArr^[3] AND 16#80) = 16#80 THEN
					pResult^ := _F_BACnet_Utf8ToWin1252(pByArr, 4);
					pBy := pBy + 4;
				END_IF
			END_IF
		END_IF
	ELSE
		(* ASCII character *)
		pResult^ := pBy^;
		pBy := pBy + 1;
	END_IF
	(* end-of-string by character *)
	IF (pResult^ = 16#00) THEN
		EXIT;
	END_IF
	(* next character *)
	pResult := pResult + 1;
	(* end-of-string by length *)
	IF (pBy >= (pString + cbString)) THEN
		EXIT;
	END_IF
END_FOR
pResult^ := 16#00;
_F_BACnet_DecodeUTF8 := pResult - pString;

END_FUNCTION

